// TwinCAT 3 PLC project plc_las_bts_vac
// ProgramVersion: 3.1.4023.0
// libraries:
//   L2SI Vacuum Library, * (SLAC)
//   LCLS General, * (SLAC)
//   PMPS, * (SLAC - LCLS)
//   Tc2_Standard, * (Beckhoff Automation GmbH)
//   Tc2_System, * (Beckhoff Automation GmbH)
//   Tc2_Utilities, * (Beckhoff Automation GmbH)
//   Tc3_Module, * (Beckhoff Automation GmbH)
// project tree:
//   DUTs/ E_TransportTube.TcDUT, ST_TransportTubeConfig.TcDUT, ST_TransportTubeDevices.TcDUT, T_TransportTube.TcDUT
//   DUTs/Operations/ E_Op.TcDUT, E_OpStep.TcDUT
//   DUTs/SystemStatusChecks/ E_GaugeCompOp.TcDUT
//   DUTs/SystemStatusChecks/Switchbox/ ST_SBGaugeReadings.TcDUT, ST_SBGaugeReadingsOp.TcDUT, ST_SBPumpStatuses.TcDUT, ST_SBValveStatuses.TcDUT
//   DUTs/SystemStatusChecks/TransportTubes/ ST_TransportTubeOps.TcDUT, ST_TransportTubeStatuses.TcDUT
//   GVLs/ GVL_BTS_VAC.TcGVL, GVL_Constants.TcGVL, GVL_MaintainLaser.TcGVL, GVL_Operation.TcGVL, GVL_TransportTubes.TcGVL
//   / PlcTask.TcTTO
//   POUs/ FB_TransportTube.TcPOU, F_UpdateIO.TcPOU, MAIN.TcPOU, MaintainLaser.TcPOU, Operate.TcPOU
//   POUs/Helpers/ F_Atm.TcPOU, F_GetTransportTube.TcPOU, F_PumpStationTurboPumpInterlock.TcPOU, F_SBVentInterlock.TcPOU
//   POUs/Operations/Abstracts/ FB_MaintainLaserOperation.TcPOU, FB_Operation.TcPOU, FB_TTOperation.TcPOU
//   POUs/Operations/ FB_LaserOn.TcPOU, FB_OpenTransportTube.TcPOU, FB_SlowPumpSwitchbox.TcPOU, FB_SlowVentSwitchbox.TcPOU, FB_VentTransportTube.TcPOU, FB_VentPumpStation.TcPOU, FB_PumpSwitchbox.TcPOU, FB_VentSwitchbox.TcPOU, FB_PumpTransportTube.TcPOU
//   POUs/Operations/MaintainLaser/ FB_SwitchboxIonPumpFailure.TcPOU, FB_SwitchboxRoughingOrTurboPumpFailure.TcPOU
//   POUs/SystemStatusChecks/ F_CompareGauge.TcPOU
//   POUs/SystemStatusChecks/Switchbox/ F_GetSBGaugeReadings.TcPOU, F_GetSBPumpStatuses.TcPOU, F_GetSBValveStatuses.TcPOU, F_SetSBPumpStatuses.TcPOU, F_SetSBValveStatuses.TcPOU, F_VerifySBGaugeReadings.TcPOU, F_VerifySBPumpStatuses.TcPOU, F_VerifySBValveStatuses.TcPOU
//   POUs/SystemStatusChecks/TransportTubes/ F_GetTransportTubeStatuses.TcPOU, F_SetTransportTubeStatuses.TcPOU, F_VerifyAllTransportTubeStatuses.TcPOU, F_VerifyTransportTubeStatuses.TcPOU (not stored)
// real-time tasks:
//   TASK PlcTask: cycle T#10ms, priority 20, ADS port 350
//   TASK OperateTask: cycle T#10ms, priority 22, ADS port 352
// I/O:
//   DEVICE =+-EK1200_00_00-CPU/EtherCAT1 (disabled), AmsNetId 5.66.246.1.2.1
//     =+-EK1200_00_00 [EK1200-5000 EtherCAT Power supply (2A E-Bus)]
//       =+-EL2794_00_01 [EL2794 4Ch. Dig. Output 24V AC/DC, 2A, short-circuit-proof]
//       =+-ES1004_00_02 [EL1004 4Ch. Dig. Input 24V, 3ms]
//       =+-ES3064_00_03 [EL3064 4Ch. Ana. Input 0-10V]
//       =+-EL1004_00_04 [EL1004 4Ch. Dig. Input 24V, 3ms]
//       =+-EL1004_00_05 [EL1004 4Ch. Dig. Input 24V, 3ms]
//       =+-EL2004_00_06 [EL2004 4Ch. Dig. Output 24V, 0.5A]
//       =+-EL1004_00_07 [EL1004 4Ch. Dig. Input 24V, 3ms]
//       =+-EL2004_00_08 [EL2004 4Ch. Dig. Output 24V, 0.5A]
//       =+-EL2004_00_09 [EL2004 4Ch. Dig. Output 24V, 0.5A]
//       =+-EL1004_00_10 [EL1004 4Ch. Dig. Input 24V, 3ms]
//       =+-EL2794_00_11 [EL2794 4Ch. Dig. Output 24V AC/DC, 2A, short-circuit-proof]
//       =+-EL1004_00_12 [EL1004 4Ch. Dig. Input 24V, 3ms]
//       =+-EL2004_00_13 [EL2004 4Ch. Dig. Output 24V, 0.5A]
//       =+-EL6021_00_14 [EL6021 Interface (RS422/485)]
//       =+-EL2202_00_15 [EL2202 2Ch. Dig. Output 24V, 0.5A]
//       =+-EL1008_00_16 [EL1008 8Ch. Dig. Input 24V, 3ms]
//       =+-EL2008_00_17 [EL2008 8Ch. Dig. Output 24V, 0.5A]
//       =+-EK1110_00_18 [EK1110 EtherCAT extension]
//     =+-EK1100_01_00 [EK1100 EtherCAT Coupler (2A E-Bus)]
//       =+-EL3174_01_18 [EL3174-0002 4Ch. Ana. Input +/-10V, +/-20mA 16 Bit, Isolated Channels]
//       =+-EL3174_01_19 [EL3174-0002 4Ch. Ana. Input +/-10V, +/-20mA 16 Bit, Isolated Channels]
//       =+-EL9184_01_20 [EL9184 Potential Connection, 8 x 24V, 8 x Ground]
//       =+-EL9070_01_21 [EL9070 Shield terminal]
//       =+-EL9070_01_22 [EL9070 Shield terminal]
//       =+-EL3174_01_23 [EL3174-0002 4Ch. Ana. Input +/-10V, +/-20mA 16 Bit, Isolated Channels]
//       =+-EL9184_01_24 [EL9184 Potential Connection, 8 x 24V, 8 x Ground]
//       =+-EL2624_01_25 [EL2624 4Ch. Relay Output, NO (125V AC / 30V DC)]
//       =+-EL2624_01_26 [EL2624 4Ch. Relay Output, NO (125V AC / 30V DC)]
//       =+-EL9505_01_27 [EL9505 Power supply terminal 5V]
//       =+-EL1124_01_28 [EL1124 4Ch. Dig. Input 5V, 10µs, Sensor Power]
//       =+-EL1124_01_29 [EL1124 4Ch. Dig. Input 5V, 10µs, Sensor Power]
//       =+-EL1124_01_30 [EL1124 4Ch. Dig. Input 5V, 10µs, Sensor Power]
//       =+-EL9410_01_31 [EL9410 E-Bus Power Supplier  (Diagnostics)]
//       =+-EL1004_01_32 [EL1004 4Ch. Dig. Input 24V, 3ms]
//       =+-EL1004_01_33 [EL1004 4Ch. Dig. Input 24V, 3ms]
//       =+-EL2794_01_34 [EL2794 4Ch. Dig. Output 24V AC/DC, 2A, short-circuit-proof]
//       =+-EK1122_01_35 [EK1122-0080 2 port EtherCAT junction (Fast Hot Connect)]
//       =+-EK1110_01_36 [EK1110 EtherCAT extension]
// variable links:
//   plc_las_bts_vac/plc_las_bts_vac Instance <-> =+-EK1200_00_00-CPU/EtherCAT1/=+-EK1100_01_00/=+-EL1124_01_28
//     PlcTask Inputs/GVL_BTS_VAC.fb_BI1_GCC.i_xDisc_Active <-> Channel 4/fb_BI1_GCC.i_xDisc_Active
//     PlcTask Inputs/GVL_BTS_VAC.fb_BI1_GCC.i_xHV_ON <-> Channel 3/fb_BI1_GCC.i_xHV_ON
//     PlcTask Inputs/GVL_BTS_VAC.fb_PP_GCC.i_xDisc_Active <-> Channel 2/fb_PP_GCC.i_xDisc_Active
//     PlcTask Inputs/GVL_BTS_VAC.fb_PP_GCC.i_xHV_ON <-> Channel 1/fb_PP_GCC.i_xHV_ON
//   plc_las_bts_vac/plc_las_bts_vac Instance <-> =+-EK1200_00_00-CPU/EtherCAT1/=+-EK1100_01_00/=+-EL1124_01_29
//     PlcTask Inputs/GVL_BTS_VAC.fb_BO4_GCC.i_xDisc_Active <-> Channel 2/fb_BO4_GCC.i_xDisc_Active
//     PlcTask Inputs/GVL_BTS_VAC.fb_BO4_GCC.i_xHV_ON <-> Channel 1/fb_BO4_GCC.i_xHV_ON
//     PlcTask Inputs/GVL_BTS_VAC.fb_DP_GCC.i_xDisc_Active <-> Channel 4/fb_DP_GCC.i_xDisc_Active
//     PlcTask Inputs/GVL_BTS_VAC.fb_DP_GCC.i_xHV_ON <-> Channel 3/fb_DP_GCC.i_xHV_ON
//   plc_las_bts_vac/plc_las_bts_vac Instance <-> =+-EK1200_00_00-CPU/EtherCAT1/=+-EK1100_01_00/=+-EL2624_01_26
//     PlcTask Outputs/GVL_BTS_VAC.fb_BI1_GCC.q_xHV_DIS <-> Channel 3/fb_BI1_GCC.q_xHV_DIS
//     PlcTask Outputs/GVL_BTS_VAC.fb_BO4_GCC.q_xHV_DIS <-> Channel 1/fb_BO4_GCC.q_xHV_DIS
//     PlcTask Outputs/GVL_BTS_VAC.fb_DP_GCC.q_xHV_DIS <-> Channel 4/fb_DP_GCC.q_xHV_DIS
//     PlcTask Outputs/GVL_BTS_VAC.fb_PP_GCC.q_xHV_DIS <-> Channel 2/fb_PP_GCC.q_xHV_DIS
//   plc_las_bts_vac/plc_las_bts_vac Instance <-> =+-EK1200_00_00-CPU/EtherCAT1/=+-EK1100_01_00/=+-EL3174_01_18
//     PlcTask Inputs/GVL_BTS_VAC.fb_BI1_GPI.i_iPRESS_R <-> AI Standard Channel 3/fb_BI1_GPI.i_iPRESS_R
//     PlcTask Inputs/GVL_BTS_VAC.fb_BO4_GPI.i_iPRESS_R <-> AI Standard Channel 1/fb_BO4_GPI.i_iPRESS_R
//     PlcTask Inputs/GVL_BTS_VAC.fb_DP_GPI.i_iPRESS_R <-> AI Standard Channel 4/fb_DP_GPI.i_iPRESS_R
//     PlcTask Inputs/GVL_BTS_VAC.fb_PP_GPI_1.i_iPRESS_R <-> AI Standard Channel 2/fb_PP_GPI_1.i_iPRESS_R
//   plc_las_bts_vac/plc_las_bts_vac Instance <-> =+-EK1200_00_00-CPU/EtherCAT1/=+-EK1100_01_00/=+-EL3174_01_19
//     PlcTask Inputs/GVL_BTS_VAC.fb_PP_GPI_2.i_iPRESS_R <-> AI Standard Channel 1/fb_PP_GPI_2.i_iPRESS_R
//   plc_las_bts_vac/plc_las_bts_vac Instance <-> =+-EK1200_00_00-CPU/EtherCAT1/=+-EK1100_01_00/=+-EL3174_01_23
//     PlcTask Inputs/GVL_BTS_VAC.fb_BI1_GCC.i_iPRESS_R <-> AI Standard Channel 3/fb_BI1_GCC.i_iPRESS_R
//     PlcTask Inputs/GVL_BTS_VAC.fb_BO4_GCC.i_iPRESS_R <-> AI Standard Channel 1/fb_BO4_GCC.i_iPRESS_R
//     PlcTask Inputs/GVL_BTS_VAC.fb_DP_GCC.i_iPRESS_R <-> AI Standard Channel 4/fb_DP_GCC.i_iPRESS_R
//     PlcTask Inputs/GVL_BTS_VAC.fb_PP_GCC.i_iPRESS_R <-> AI Standard Channel 2/fb_PP_GCC.i_iPRESS_R
//   plc_las_bts_vac/plc_las_bts_vac Instance <-> =+-EK1200_00_00-CPU/EtherCAT1/=+-EK1200_00_00/=+-EL1004_00_04
//     PlcTask Inputs/GVL_BTS_VAC.fb_BI1_VGC.i_xClsLS <-> Channel 1/fb_BI1_VGC.i_xClsLS
//     PlcTask Inputs/GVL_BTS_VAC.fb_BI1_VGC.i_xOpnLS <-> Channel 2/fb_BI1_VGC.i_xOpnLS
//     PlcTask Inputs/GVL_BTS_VAC.fb_BO4_VGC.i_xClsLS <-> Channel 3/fb_BO4_VGC.i_xClsLS
//     PlcTask Inputs/GVL_BTS_VAC.fb_BO4_VGC.i_xOpnLS <-> Channel 4/fb_BO4_VGC.i_xOpnLS
//   plc_las_bts_vac/plc_las_bts_vac Instance <-> =+-EK1200_00_00-CPU/EtherCAT1/=+-EK1200_00_00/=+-EL1004_00_05
//     PlcTask Inputs/GVL_BTS_VAC.fb_PP_VGC.i_xClsLS <-> Channel 3/fb_PP_VGC.i_xClsLS
//     PlcTask Inputs/GVL_BTS_VAC.fb_PP_VGC.i_xOpnLS <-> Channel 4/fb_PP_VGC.i_xOpnLS
//     PlcTask Inputs/GVL_BTS_VAC.fb_PP_VRC_1.i_xClsLS <-> Channel 1/fb_PP_VRC_1.i_xClsLS
//     PlcTask Inputs/GVL_BTS_VAC.fb_PP_VRC_1.i_xOpnLS <-> Channel 2/fb_PP_VRC_1.i_xOpnLS
//   plc_las_bts_vac/plc_las_bts_vac Instance <-> =+-EK1200_00_00-CPU/EtherCAT1/=+-EK1200_00_00/=+-EL1004_00_07
//     PlcTask Inputs/GVL_BTS_VAC.fb_PP_VRC_2.i_xClsLS <-> Channel 1/fb_PP_VRC_2.i_xClsLS
//     PlcTask Inputs/GVL_BTS_VAC.fb_PP_VRC_3.i_xClsLS <-> Channel 3/fb_PP_VRC_3.i_xClsLS
//     PlcTask Inputs/GVL_BTS_VAC.fb_PP_VRC_2.i_xOpnLS <-> Channel 2/fb_PP_VRC_2.i_xOpnLS
//     PlcTask Inputs/GVL_BTS_VAC.fb_PP_VRC_3.i_xOpnLS <-> Channel 4/fb_PP_VRC_3.i_xOpnLS
//   plc_las_bts_vac/plc_las_bts_vac Instance <-> =+-EK1200_00_00-CPU/EtherCAT1/=+-EK1200_00_00/=+-EL1004_00_10
//     PlcTask Inputs/GVL_BTS_VAC.fb_PP_PMF.i_xAlarm <-> Channel 3/fb_PP_PMF.i_xAlarm
//     PlcTask Inputs/GVL_BTS_VAC.fb_PP_PMF.i_xIsRun <-> Channel 1/fb_PP_PMF.i_xIsRun
//     PlcTask Inputs/GVL_BTS_VAC.fb_PP_PMF.i_xLocal <-> Channel 2/fb_PP_PMF.i_xLocal
//     PlcTask Inputs/GVL_BTS_VAC.fb_PP_PMF.i_xWarning <-> Channel 4/fb_PP_PMF.i_xWarning
//   plc_las_bts_vac/plc_las_bts_vac Instance <-> =+-EK1200_00_00-CPU/EtherCAT1/=+-EK1200_00_00/=+-EL1004_00_12
//     PlcTask Inputs/GVL_BTS_VAC.fb_PP_PTM.i_xAtSpd <-> Channel 1/fb_PP_PTM.i_xAtSpd
//     PlcTask Inputs/GVL_BTS_VAC.fb_PP_PTM.i_xFaultNC <-> Channel 3/fb_PP_PTM.i_xFaultNC
//     PlcTask Inputs/GVL_BTS_VAC.fb_PP_PTM.i_xRemote <-> Channel 2/fb_PP_PTM.i_xRemote
//   plc_las_bts_vac/plc_las_bts_vac Instance <-> =+-EK1200_00_00-CPU/EtherCAT1/=+-EK1200_00_00/=+-EL2004_00_06
//     PlcTask Outputs/GVL_BTS_VAC.fb_BI1_VGC.q_xOPN_DO <-> Channel 1/fb_BI1_VGC.q_xOPN_DO
//     PlcTask Outputs/GVL_BTS_VAC.fb_BO4_VGC.q_xOPN_DO <-> Channel 3/fb_BO4_VGC.q_xOPN_DO
//   plc_las_bts_vac/plc_las_bts_vac Instance <-> =+-EK1200_00_00-CPU/EtherCAT1/=+-EK1200_00_00/=+-EL2004_00_08
//     PlcTask Outputs/GVL_BTS_VAC.fb_PP_VGC.q_xOPN_DO <-> Channel 2/fb_PP_VGC.q_xOPN_DO
//     PlcTask Outputs/GVL_BTS_VAC.fb_PP_VRC_1.q_xOPN_DO <-> Channel 1/fb_PP_VRC_1.q_xOPN_DO
//     PlcTask Outputs/GVL_BTS_VAC.fb_PP_VRC_2.q_xOPN_DO <-> Channel 3/fb_PP_VRC_2.q_xOPN_DO
//     PlcTask Outputs/GVL_BTS_VAC.fb_PP_VRC_3.q_xOPN_DO <-> Channel 4/fb_PP_VRC_3.q_xOPN_DO
//   plc_las_bts_vac/plc_las_bts_vac Instance <-> =+-EK1200_00_00-CPU/EtherCAT1/=+-EK1200_00_00/=+-EL2004_00_09
//     PlcTask Outputs/GVL_BTS_VAC.fb_PP_VVC.q_xOPN_DO <-> Channel 3/fb_PP_VVC.q_xOPN_DO
//     PlcTask Outputs/GVL_BTS_VAC.fb_VP_VVC_1.xCLS_DO <-> Channel 1/fb_VP_VVC_1.xCLS_DO
//     PlcTask Outputs/GVL_BTS_VAC.fb_VP_VVC_2.xCLS_DO <-> Channel 2/fb_VP_VVC_2.xCLS_DO
//   plc_las_bts_vac/plc_las_bts_vac Instance <-> =+-EK1200_00_00-CPU/EtherCAT1/=+-EK1200_00_00/=+-EL2004_00_13
//     PlcTask Outputs/GVL_BTS_VAC.fb_PP_PTM.q_PumpingStation <-> Channel 3/fb_PP_PTM.q_PumpingStation
//     PlcTask Outputs/GVL_BTS_VAC.fb_PP_PTM.q_RunDO <-> Channel 1/fb_PP_PTM.q_RunDO
//     PlcTask Outputs/GVL_BTS_VAC.fb_PP_PTM.q_xRemote <-> Channel 2/fb_PP_PTM.q_xRemote
//   plc_las_bts_vac/plc_las_bts_vac Instance <-> =+-EK1200_00_00-CPU/EtherCAT1/=+-EK1200_00_00/=+-EL2794_00_01
//     PlcTask Outputs/GVL_BTS_VAC.fb_BI1_PIP.q_xHVEna_DO <-> Channel 2/fb_BI1_PIP.q_xHVEna_DO
//     PlcTask Outputs/GVL_BTS_VAC.fb_BO4_PIP.q_xHVEna_DO <-> Channel 1/fb_BO4_PIP.q_xHVEna_DO
//     PlcTask Outputs/GVL_BTS_VAC.fb_PP_PIP.q_xHVEna_DO <-> Channel 3/fb_PP_PIP.q_xHVEna_DO
//   plc_las_bts_vac/plc_las_bts_vac Instance <-> =+-EK1200_00_00-CPU/EtherCAT1/=+-EK1200_00_00/=+-EL2794_00_11
//     PlcTask Outputs/GVL_BTS_VAC.fb_PP_PMF.q_xLspdDo <-> Channel 2/fb_PP_PMF.q_xLspdDo
//     PlcTask Outputs/GVL_BTS_VAC.fb_PP_PMF.q_xResetDo <-> Channel 3/fb_PP_PMF.q_xResetDo
//     PlcTask Outputs/GVL_BTS_VAC.fb_PP_PMF.q_xRunDO <-> Channel 1/fb_PP_PMF.q_xRunDO
//   plc_las_bts_vac/plc_las_bts_vac Instance <-> =+-EK1200_00_00-CPU/EtherCAT1/=+-EK1200_00_00/=+-ES1004_00_02
//     PlcTask Inputs/GVL_BTS_VAC.fb_BI1_PIP.i_xSP_DI <-> Channel 2/fb_BI1_PIP.i_xSP_DI
//     PlcTask Inputs/GVL_BTS_VAC.fb_BO4_PIP.i_xSP_DI <-> Channel 1/fb_BO4_PIP.i_xSP_DI
//     PlcTask Inputs/GVL_BTS_VAC.fb_PP_PIP.i_xSP_DI <-> Channel 3/fb_PP_PIP.i_xSP_DI
//   plc_las_bts_vac/plc_las_bts_vac Instance <-> =+-EK1200_00_00-CPU/EtherCAT1/=+-EK1200_00_00/=+-ES3064_00_03
//     PlcTask Inputs/GVL_BTS_VAC.fb_BI1_PIP.i_iPRESS <-> AI Standard Channel 2/fb_BI1_PIP.i_iPRESS
//     PlcTask Inputs/GVL_BTS_VAC.fb_BO4_PIP.i_iPRESS <-> AI Standard Channel 1/fb_BO4_PIP.i_iPRESS
//     PlcTask Inputs/GVL_BTS_VAC.fb_PP_PIP.i_iPRESS <-> AI Standard Channel 3/fb_PP_PIP.i_iPRESS

CONFIGURATION plc_las_bts_vac
    RESOURCE PLC ON TwinCAT3
        TASK PlcTask(INTERVAL := T#10ms, PRIORITY := 20);
        PROGRAM MAIN WITH PlcTask : MAIN;
        PROGRAM Operate WITH PlcTask : Operate;
        PROGRAM MaintainLaser WITH PlcTask : MaintainLaser;
    END_RESOURCE
END_CONFIGURATION

// ---- DUTs/E_TransportTube.TcDUT
{attribute 'qualified_only'}
TYPE E_TransportTube :
(
	LS1 := 0,
	LS5 := 1,
	LS8 := 2,
	LD2 := 3,
	LD4 := 4,
	LD6 := 5,
	LD8 := 6,
	LD9 := 7,
	LD10 := 8,
	LD14 := 9
) UINT;
END_TYPE

// ---- DUTs/Operations/E_Op.TcDUT
{attribute 'qualified_only'}
{attribute 'strict'}
TYPE E_Op :
(
	NONE := 0, // No operation
	PSB := 1, // Pump switchbox
	VSB := 2, // Vent switchbox
	VPS := 3, // Vent pumping station
	PTT := 4, // Transport tube pump down
	VTT := 5, // Transport tube vent
	LTT := 6, // Turn on laser for transport tube
	SPSB := 7, // Slow Pump Switchbox
	SVSB := 8 // Slow Vent switchbox
	//OTT, // Open transport tube gate valve
);
END_TYPE

// ---- DUTs/Operations/E_OpStep.TcDUT
{attribute 'qualified_only'}
{attribute 'strict'}
TYPE E_OpStep :
(
	IDLE := 0,
	START := 1,
	
	(* Pump Switchbox steps *)
	PSB_OPEN_GATE_VALVE,
	PSB_OPEN_PUMP_STATION_VALVES,
	PSB_ROUGH_CHAMBER,
	PSB_TURBO_CHAMBER,
	PSB_SWITCH_TO_ION_PUMP,
	PSB_CLOSE_GATE_VALVE,
	PSB_STOP_TURBO_PUMP,
	PSB_FINISH,
	
	(* Slow Pump switchbox steps *)
	SPSB_OPEN_GATE_VALVE,
	SPSB_OPEN_PUMP_STATION_VALVES,
	SPSB_ROUGH_CHAMBER,
	SPSB_OPEN_FORELINE_VALVE,
	SPSB_TURBO_CHAMBER,
	SPSB_SWITCH_TO_ION_PUMP,
	SPSB_CLOSE_VALVES,
	SPSB_STOP_TURBO_PUMP,
	SPSB_FINISH,
	
	(* Vent Switchbox steps *)
	VSB_CLOSE_GATE_VALVE,
	VSB_CLOSE_FORELINE_VALVE,
	VSB_TURN_OFF_PUMPS,
	VSB_CLOSE_ORING_VALVE,
	VSB_VENT,
	VSB_CLOSE_VENT,
	VSB_FINISH,
	
	(* Slow Vent Switchbox steps *)
	SVSB_CLOSE_GATE_VALVE,
	SVSB_CLOSE_FORELINE_VALVE,
	SVSB_TURN_OFF_PUMPS,
	SVSB_CLOSE_ORING_VALVE,
	SVSB_VENT,
	SVSB_SLOW_VENT,
	SVSB_CLOSE_VENT,
	SVSB_FINISH,
	
	(* Vent pump station *)
	VPS_VENT,
	VPS_CLOSE_VENT,
	VPS_FINISH,
	
	(* Pump Down Transport Tube *)
	POT_WAIT_PUMP_CART,
	POT_TURN_ON_PUMP,
	POT_FINISH,
	
	(* Vent Transport Tube *)
	VOT_VENT,
	VOT_WAIT_PC,
	VOT_FINISH,
	
	(* Open Transport Tube Gate Valve *)
	OTT_OPEN_VALVE,
	OTT_RUN_PSB,
	OTT_RUN_PTT,
	
	(* Laser Transport Tube On *)
	LTT_RUN_PSB,
	LTT_RUN_PTT,
	
	(* Beam On - Switchbox Ion Pump Failure *)
	BOIP_TURN_OFF_ION_PUMP,
	BOIP_OPEN_SB_VALVE,
	BOIP_HOLD,
	BOIP_CLOSE_TRANSPORT_TUBE_VALVES,
	BOIP_CLOSE_SB_VALVE,
	BOIP_TURN_OFF_PUMPS,
	BOIP_CLOSE_PP_VALVES,
	BOIP_VENT_SB,
	
	(* Beam On - Switchbox Roughing Pump or Turbo Pump Failure *)
	BOPL_TURN_ON_ION_PUMP,
	BOPL_CLOSE_PP_VALVES,
	BOPL_TURN_OFF_PP_PUMPS,
	BOPL_HOLD,
	BOPL_CLOSE_TRANSPORT_TUBE_VALVES,
	BOPL_VENT_SB
);
END_TYPE

// ---- DUTs/ST_TransportTubeConfig.TcDUT
TYPE ST_TransportTubeConfig :
STRUCT
	{attribute 'pytmc' := '
		pv: NAME
		io: i
	'}
	sName : STRING(EPICS_STRING_SIZE);
	
	bInput : BOOL; // True for input tube, false for output tube
	
	stDevices : ST_TransportTubeDevices;
END_STRUCT
END_TYPE

// ---- DUTs/ST_TransportTubeDevices.TcDUT
(* Devices common to all transport tubes. *)
TYPE ST_TransportTubeDevices :
STRUCT
	// Pumps
	refIonPump : REFERENCE TO FB_PIP_GAMMA;
	
	// Valves
	refGateValve : REFERENCE TO FB_VGC;
	
	// Gauges
	refPiraniGauge : REFERENCE TO FB_MKS275;
	refColdCathode : REFERENCE TO FB_MKS500;
END_STRUCT
END_TYPE

// ---- DUTs/SystemStatusChecks/E_GaugeCompOp.TcDUT
(* Comparison operators that can be used to compare gauge readings *)
{attribute 'qualified_only'}
{attribute 'strict'}
TYPE E_GaugeCompOp :
(
	IGNORE, // Ignore the gauge reading
	ATM, // Check that gauge is at atmospheric pressure
	_LTE, // Check that gauge is less than or equal to value
	_GTE, // Check that gauge is greater than or equal to value
	STATE // Check that gauge has a specific state
):= IGNORE;
END_TYPE

// ---- DUTs/SystemStatusChecks/Switchbox/ST_SBGaugeReadings.TcDUT
(* Statuses of the gauges for the switchbox *)
TYPE ST_SBGaugeReadings :
STRUCT
	(* Gauge readings *)
	
	fDPPiraniVal : REAL; // LXLHN:DP:GPI
	eDPPiraniState : E_PressureState;
	
	fDPColdCathodeVal : REAL; // LXLHN:DP:GCC
	eDPColdCathodeState : E_PressureState;
	
	fPumpStationPirani1Val : REAL; // LXLHN:PP:GPI:1
	ePumpStationPirani1State : E_PressureState;
	
	fPumpStationPirani2Val : REAL; // LXLHN:PP:GPI:2
	ePumpStationPirani2State : E_PressureState;
	
	fPumpStationColdCathodeVal : REAL; // LXLHN:PP:GCC
	ePumpStationColdCathodeState : E_PressureState;
END_STRUCT
END_TYPE

// ---- DUTs/SystemStatusChecks/Switchbox/ST_SBGaugeReadingsOp.TcDUT
(* What operations should be used to compare gauge status *)
TYPE ST_SBGaugeReadingsOp :
STRUCT
	eDPPiraniOp : E_GaugeCompOp; // LXLHN:DP:GPI
	eDPColdCathodeOp : E_GaugeCompOp; // LXLHN:DP:GCC
	ePumpStationPirani1Op : E_GaugeCompOp; // LXLHN:PP:GPI:1
	ePumpStationPirani2Op : E_GaugeCompOp; // LXLHN:PP:GPI:2
	ePumpStationColdCathodeOp : E_GaugeCompOp; // LXLHN:PP:GCC
END_STRUCT
END_TYPE

// ---- DUTs/SystemStatusChecks/Switchbox/ST_SBPumpStatuses.TcDUT
(* Statuses of the pumps for the switchbox *)
TYPE ST_SBPumpStatuses :
STRUCT
	// Pump statuses
	bRoughingPumpOn : BOOL; // LXLHN:PP:PMF
	bTurboPumpOn : BOOL; // LXLHN:PP:PTM
	bIonPumpOn : BOOL; // LXLHN:PP:PIP
END_STRUCT
END_TYPE

// ---- DUTs/SystemStatusChecks/Switchbox/ST_SBValveStatuses.TcDUT
(* Statuses of the valves for the switchbox *)
TYPE ST_SBValveStatuses :
STRUCT
	// Valve statuses
	bGateValveOpen : BOOL; // LXLHN:PP:VGC
	bVentValveOpen : BOOL; // LXLHN:PP:VVC
	bORingPumpValveOpen : BOOL; // LXLHN:PP:VRC:1
	bForelineValveOpen : BOOL; // LXLHN:PP:VRC:2
	bSlowPumpValveOpen : BOOL; // LXLHN:PP:VRC:3
	bSBVentOpen : BOOL; // LXLHN:VP:VVC1
	bSBSlowVentOpen : BOOL; // LXLHN:VP:VVC:2
END_STRUCT
END_TYPE

// ---- DUTs/SystemStatusChecks/TransportTubes/ST_TransportTubeOps.TcDUT
TYPE ST_TransportTubeOps :
STRUCT
	// Pumps
	bIonPumpIgnore : BOOL := FALSE;
	
	// Valves
	bGateValveIgnore : BOOL := FALSE;
	
	// Gauges
	ePiraniOp : E_GaugeCompOp := E_GaugeCompOp.IGNORE;
	eColdCathodeOp : E_GaugeCompOp := E_GaugeCompOp.IGNORE;
END_STRUCT
END_TYPE

// ---- DUTs/SystemStatusChecks/TransportTubes/ST_TransportTubeStatuses.TcDUT
(* Statuses of the pumps, valves, and gauges for the for the BO4 Output tube *)
TYPE ST_TransportTubeStatuses :
STRUCT
	// Pump statuses
	bIonPumpOn : BOOL;
	
	// Valve statuses
	bGateValveOpen : BOOL;
	
	// Gauge statuses
	fPiraniVal : REAL;
	ePiraniState : E_PressureState;
	fColdCathodeVal : REAL;
	eColdCathodeState : E_PressureState;
	
END_STRUCT
END_TYPE

// ---- DUTs/T_TransportTube.TcDUT
// Create a generic transport tube type in case E_TransportTube ever needs to be split up into
// multiple enums (such as input and output tubes). That way all the different Transport tube enums 
// can still have a common type.
TYPE T_TransportTube : UINT; END_TYPE

// ---- GVLs/GVL_BTS_VAC.TcGVL
{attribute 'qualified_only'}
VAR_GLOBAL
	(* Valves *)	
	fb_PP_VGC_FFOut : FB_HardwareFFOutput;
	{attribute 'pytmc' := 'pv: LXLHN:PP:VGC'}
	fb_PP_VGC : FB_VGC; // Gate valve, vacuum switchbox
	
	{attribute 'pytmc' := 'pv: LXLHN:PP:VVC'}
	fb_PP_VVC : FB_VVC; // Turbo N2 purge
	
	{attribute 'pytmc' := 'pv: LXLHN:PP:VRC:1'}
	fb_PP_VRC_1 : FB_VRC; // O-ring diff pump valve
	
	{attribute 'pytmc' := 'pv: LXLHN:PP:VRC:2'}
	fb_PP_VRC_2 : FB_VRC; // Foreline valve
	
	{attribute 'pytmc' := 'pv: LXLHN:PP:VRC:3'}
	fb_PP_VRC_3 : FB_VRC; // Slow pump valve
	
	st_VP_VVC_1 : ST_VCC_NO;
	{attribute 'pytmc' := 'pv: LXLHN:VP:VVC:1'}
	fb_VP_VVC_1 : FB_VCC_NO; // Vent valve, Switchbox
	
	st_VP_VVC_2 : ST_VCC_NO;
	{attribute 'pytmc' := 'pv: LXLHN:VP:VVC:2'}
	fb_VP_VVC_2 : FB_VCC_NO; // Vent valve, Slow, Switchbox

	
	(* Pumps *)
	{attribute 'pytmc' := 'pv: LXLHN:PP:PTM'}
	fb_PP_PTM : FB_PTM_Pfeiffer; // Turbo pump
	
	{attribute 'pytmc' := 'pv: LXLHN:PP:PMF'}
	fb_PP_PMF : FB_KashiyamaPump; // Roughing Pump
	
	{attribute 'pytmc' := 'pv: LXLHN:PP:PIP'}
	fb_PP_PIP : FB_PIP_Gamma; // Ion Pump, SW
	
	(* Gauges *)
	{attribute 'pytmc' := 'pv: LXLHN:PP:GPI:1'}
	fb_PP_GPI_1 : FB_MKS275; // Switchbox pumpline ATM gauge
	
	{attribute 'pytmc' := 'pv: LXLHN:PP:GPI:2'}
	fb_PP_GPI_2 : FB_MKS275; // Foreline gauge
	
	{attribute 'pytmc' := 'pv: LXLHN:DP:GPI'}
	fb_DP_GPI : FB_MKS275; // Switchbox gauge
	
	{attribute 'pytmc' := 'pv: LXLHN:PP:GCC'}
	fb_PP_GCC : FB_MKS500; // Switchbox pumpline Cold Cathode gauge
	
	{attribute 'pytmc' := 'pv: LXLHN:DP:GCC'}
	fb_DP_GCC : FB_MKS500; // Switchbox Cold Cathode gauge
	
	(* Transport Tubes *)
	// LS1
	fb_LS1_VGC_FFOut : FB_HardwareFFOutput;
	{attribute 'pytmc' := 'pv: LTLHN:LS1:VGC:01'}
	fb_LS1_VGC : FB_VGC; // Gate valve, Input LS1 laser Table
	{attribute 'pytmc' := 'pv: LTLHN:LS1:PIP:01'}
	fb_LS1_PIP : FB_PIP_Gamma; // Ion Pump, input tube LS1
	{attribute 'pytmc' := 'pv: LTLHN:LS1:GPI:01'}
	fb_LS1_GPI : FB_MKS275; // Input tube LS1 ATM gauge
	{attribute 'pytmc' := 'pv: LTLHN:LS1:GCC:01'}
	fb_LS1_GCC : FB_MKS500; // Input tube LS1, Cold Cathode gauge
	
	// LS5
	fb_LS5_VGC_FFOut : FB_HardwareFFOutput;
	{attribute 'pytmc' := 'pv: LTLHN:LS5:VGC:01'}
	fb_LS5_VGC : FB_VGC; // Gate valve, Input LS5 laser Table
	{attribute 'pytmc' := 'pv: LTLHN:LS5:PIP:01'}
	fb_LS5_PIP : FB_PIP_Gamma; // Ion Pump, input tube LS5
	{attribute 'pytmc' := 'pv: LTLHN:LS5:GPI:01'}
	fb_LS5_GPI : FB_MKS275; // Input tube LS5 ATM gauge
	{attribute 'pytmc' := 'pv: LTLHN:LS5:GCC:01'}
	fb_LS5_GCC : FB_MKS500; // Input tube LS5, Cold Cathode gauge
	
	// LS8
	fb_LS8_VGC_FFOut : FB_HardwareFFOutput;
	{attribute 'pytmc' := 'pv: LTLHN:LS8:VGC:01'}
	fb_LS8_VGC : FB_VGC; // Gate valve, Input LS8 laser Table
	{attribute 'pytmc' := 'pv: LTLHN:LS8:PIP:01'}
	fb_LS8_PIP : FB_PIP_Gamma; // Ion Pump, input tube LS8
	{attribute 'pytmc' := 'pv: LTLHN:LS8:GPI:01'}
	fb_LS8_GPI : FB_MKS275; // Input tube LS8 ATM gauge
	{attribute 'pytmc' := 'pv: LTLHN:LS8:GCC:01'}
	fb_LS8_GCC : FB_MKS500; // Input tube LS8, Cold Cathode gauge

	// LD2
	fb_LD2_VGC_FFOut : FB_HardwareFFOutput;
	{attribute 'pytmc' := 'pv: LTLHN:LD2:VGC:01'}
	fb_LD2_VGC : FB_VGC; // Gate valve, Output tube LD2 laser Table
	{attribute 'pytmc' := 'pv: LTLHN:LD2:PIP:01'}
	fb_LD2_PIP : FB_PIP_Gamma; // Ion Pump, output tube LD2
	{attribute 'pytmc' := 'pv: LTLHN:LD2:GPI:01 '}
	fb_LD2_GPI : FB_MKS275; // Output tube LD2 ATM gauge
	{attribute 'pytmc' := 'pv: LTLHN:LD2:GCC:01'}
	fb_LD2_GCC : FB_MKS500; // Output tube LD2, Cold Cathode gauge
	
	// LD4
	fb_LD4_VGC_FFOut : FB_HardwareFFOutput;
	{attribute 'pytmc' := 'pv: LTLHN:LD4:VGC:01'}
	fb_LD4_VGC : FB_VGC; // Gate valve, Output tube LD4 laser Table
	{attribute 'pytmc' := 'pv: LTLHN:LD4:PIP:01'}
	fb_LD4_PIP : FB_PIP_Gamma; // Ion Pump, output tube LD4
	{attribute 'pytmc' := 'pv: LTLHN:LD4:GPI:01'}
	fb_LD4_GPI : FB_MKS275; // Output tube LD4 ATM gauge
	{attribute 'pytmc' := 'pv: LTLHN:LD4:GCC:01'}
	fb_LD4_GCC : FB_MKS500; // Output tube LD4, Cold Cathode gauge
	
	// LD6
	fb_LD6_VGC_FFOut : FB_HardwareFFOutput;
	{attribute 'pytmc' := 'pv: LTLHN:LD6:VGC:01'}
	fb_LD6_VGC : FB_VGC; // Gate valve, Output tube LD6 laser Table
	{attribute 'pytmc' := 'pv: LTLHN:LD6:PIP:01'}
	fb_LD6_PIP : FB_PIP_Gamma; // Ion Pump, output tube LD6
	{attribute 'pytmc' := 'pv: LTLHN:LD6:GPI:01'}
	fb_LD6_GPI : FB_MKS275; // Output tube LD6 ATM gauge
	{attribute 'pytmc' := 'pv: LTLHN:LD6:GCC:01'}
	fb_LD6_GCC : FB_MKS500; // Output tube LD6, Cold Cathode gauge
	
	// LD14
	fb_LD14_VGC_FFOut : FB_HardwareFFOutput;
	{attribute 'pytmc' := 'pv: LTLHN:LD14:VGC:01'}
	fb_LD14_VGC : FB_VGC; // Gate valve, Output tube LD14 laser Table
	{attribute 'pytmc' := 'pv: LTLHN:LD14:PIP:01'}
	fb_LD14_PIP : FB_PIP_Gamma; // Ion Pump, output tube LD14
	{attribute 'pytmc' := 'pv: LTLHN:LD14:GPI:01'}
	fb_LD14_GPI : FB_MKS275; // Output tube LD14 ATM gauge
	{attribute 'pytmc' := 'pv: LTLHN:LD14:GCC:01'}
	fb_LD14_GCC : FB_MKS500; // Output tube LD14, Cold Cathode gauge
	
	// LD10
	fb_LD10_VGC_FFOut : FB_HardwareFFOutput;
	{attribute 'pytmc' := 'pv: LTLHN:LD10:VGC:01'}
	fb_LD10_VGC : FB_VGC; // Gate valve, Output tube LD10 laser Table
	{attribute 'pytmc' := 'pv: LTLHN:LD10:PIP:01'}
	fb_LD10_PIP : FB_PIP_Gamma; // Ion Pump, output tube LD10
	{attribute 'pytmc' := 'pv: LTLHN:LD10:GPI:01'}
	fb_LD10_GPI : FB_MKS275; // Output tube LD10 ATM gauge
	{attribute 'pytmc' := 'pv: LTLHN:LD10:GCC:01'}
	fb_LD10_GCC : FB_MKS500; // Output tube LD10, Cold Cathode gauge
	
	// LD9
	fb_LD9_VGC_FFOut : FB_HardwareFFOutput;
	{attribute 'pytmc' := 'pv: LTLHN:LD9:VGC:01'}
	fb_LD9_VGC : FB_VGC; // Gate valve, Output tube LD9 laser Table
	{attribute 'pytmc' := 'pv: LTLHN:LD9:PIP:01'}
	fb_LD9_PIP : FB_PIP_Gamma; // Ion Pump, output tube LD9
	{attribute 'pytmc' := 'pv: LTLHN:LD9:GPI:01'}
	fb_LD9_GPI : FB_MKS275; // Output tube LD9 ATM gauge
	{attribute 'pytmc' := 'pv: LTLHN:LD9:GCC:01'}
	fb_LD9_GCC : FB_MKS500; // Output tube LD9, Cold Cathode gauge
	
	// LD8
	fb_LD8_VGC_FFOut : FB_HardwareFFOutput;
	{attribute 'pytmc' := 'pv: LTLHN:LD8:VGC:01'}
	fb_LD8_VGC : FB_VGC; // Gate valve, Output tube LD8 laser Table
	{attribute 'pytmc' := 'pv: LTLHN:LD8:PIP:01'}
	fb_LD8_PIP : FB_PIP_Gamma; // Ion Pump, output tube LD8
	{attribute 'pytmc' := 'pv: LTLHN:LD8:GPI:01'}
	fb_LD8_GPI : FB_MKS275; // Output tube LD8 ATM gauge
	{attribute 'pytmc' := 'pv: LTLHN:LD8:GCC:01'}
	fb_LD8_GCC : FB_MKS500; // Output tube LD8, Cold Cathode gauge

END_VAR

// ---- GVLs/GVL_Constants.TcGVL
VAR_GLOBAL CONSTANT
	ATM_PRESS : INT := 760; // Atmospheric pressure in Torr
	ATM_PRESS_ERR_RNG : INT := 10; // Error range that is still considered atmospheric pressure
	
	EPICS_STRING_SIZE : INT := 40;
	PTM_INTERLOCK_SP : REAL := 1E-2;
END_VAR

// ---- GVLs/GVL_MaintainLaser.TcGVL
{attribute 'qualified_only'}
VAR_GLOBAL
	{attribute 'pytmc' := '
		pv: PLC_LAS_BTS_VAC:LASER_MAINTAINER:BUSY
		io: i
		field: ZNAM NOT_BUSY
		field: ONAM BUSY
	'}
	q_bOperationInProgress : BOOL;
	
	{attribute 'pytmc' := '
		pv: PLC_LAS_BTS_VAC:LASER_MAINTAINER:RESET
		io: o
	'}
	i_bReset : BOOL; // Reset the laser maintainer to default state
	
	{attribute 'pytmc' := '
		pv: PLC_LAS_BTS_VAC:LASER_MAINTAINER:SHUTOFF
		io: o		
	'}
	i_bShutoff : BOOL; // Signal to shutoff all laser ok signals
	
	{attribute 'pytmc' := '
		pv: PLC_LAS_BTS_VAC:LASER_MAINTAINER:ION_PUMP_FAILURE
		io: i
		field: ZNAM OK
		field: ONAM ERROR
		field: OSV MAJOR
	'}
	q_bIonPumpFailure : BOOL;
	
	{attribute 'pytmc' := '
		pv: PLC_LAS_BTS_VAC:LASER_MAINTAINER:TURBO_PUMP_FAILURE
		io: i
		field: ZNAM OK
		field: ONAM ERROR
		field: OSV MAJOR
	'}
	q_bTurboPumpFailure : BOOL;
	
	{attribute 'pytmc' := '
		pv: PLC_LAS_BTS_VAC:LASER_MAINTAINER:ROUGHING_PUMP_FAILURE
		io: i
		field: ZNAM OK
		field: ONAM ERROR
		field: OSV MAJOR
	'}
	q_bRoughingPumpFailure : BOOL;
	
	{attribute 'pytmc' := '
		pv: PLC_LAS_BTS_VAC:LASER_MAINTAINER:MESSAGE
		io: i
	'}
	q_sMessage : STRING(EPICS_STRING_SIZE) := 'No issues';
	
	{attribute 'pytmc' := '
		pv: PLC_LAS_BTS_VAC:LASER_MAINTAINER:SHUTOFF_LATCH
		io: i
		field: ZNAM OK
		field: ONAM LASERS_SHUTOFF
		field: OSV MAJOR
	'}
	q_bShutoffLatch : BOOL;
END_VAR

// ---- GVLs/GVL_Operation.TcGVL
{attribute 'qualified_only'}
VAR_GLOBAL
	// Execute flags for vacuum system operations
	{attribute 'pytmc' := '
		pv: PLC_LAS_BTS_VAC:OPERATION:CANCEL
		io: o
	'}
	i_bCancel : BOOL;
	
	{attribute 'pytmc' := '
		pv: PLC_LAS_BTS_VAC:OPERATION
		io: io
	'}
	iq_eOperation : E_Op;
	
	{attribute 'pytmc' := '
		pv: PLC_LAS_BTS_VAC:OPERATION:TRANSPORT_TUBE
		io: io
	'}
	iq_eTransportTube : E_TransportTube;
	
	{attribute 'pytmc' := '
		pv: PLC_LAS_BTS_VAC:OPERATION:BUSY
		io: i
		field: ZNAM NOT_BUSY
		field: ONAM BUSY
	'}
	q_bBusy : BOOL;
	
	{attribute 'pytmc' := '
		pv: PLC_LAS_BTS_VAC:OPERATION:ERROR
		io: i
		field: ZNAM OK
		field: ONAM ERROR
		field: ZSV NO_ALARM
		field: OSV MAJOR
	'}
	q_bError : BOOL;
	
	{attribute 'pytmc' := '
		pv: PLC_LAS_BTS_VAC:OPERATION:MESSAGE
		io: i
	'}
	q_sMessage : STRING(EPICS_STRING_SIZE);
END_VAR

// ---- GVLs/GVL_TransportTubes.TcGVL
{attribute 'qualified_only'}
VAR_GLOBAL CONSTANT
	// When adding transport tubes make sure to update F_GetTransportTube!
	
	NUM_TRANSPORT_TUBES : UINT := 10;
	
	aTubes : ARRAY [1..NUM_TRANSPORT_TUBES] OF T_TransportTube := [
		(* Input transport tubes *)
		E_TransportTube.LS1,
		E_TransportTube.LS5,
		E_TransportTube.LS8, 
		
		(* Output transport tubes *)
		E_TransportTube.LD2,
		E_TransportTube.LD4,
		E_TransportTube.LD6,
		E_TransportTube.LD8,
		E_TransportTube.LD9,
		E_TransportTube.LD10,
		E_TransportTube.LD14
	];
	
	(* Transport tube configs *)
	
	stLS1 : ST_TransportTubeConfig := (
		sName:= 'LS1',
		bInput := TRUE,
		stDevices:= (
			refIonPump := GVL_BTS_VAC.fb_LS1_PIP,
			refGateValve := GVL_BTS_VAC.fb_LS1_VGC,
			refPiraniGauge := GVL_BTS_VAC.fb_LS1_GPI,
			refColdCathode := GVL_BTS_VAC.fb_LS1_GCC)
	);
	
	stLS5 : ST_TransportTubeConfig := (
		sName:= 'LS5',
		bInput := TRUE,
		stDevices:= (
			refIonPump := GVL_BTS_VAC.fb_LS5_PIP,
			refGateValve := GVL_BTS_VAC.fb_LS5_VGC,
			refPiraniGauge := GVL_BTS_VAC.fb_LS5_GPI,
			refColdCathode := GVL_BTS_VAC.fb_LS5_GCC)
	);
	
	stLS8 : ST_TransportTubeConfig := (
		sName:= 'LS8',
		bInput := TRUE,
		stDevices:= (
			refIonPump := GVL_BTS_VAC.fb_LS8_PIP,
			refGateValve := GVL_BTS_VAC.fb_LS8_VGC,
			refPiraniGauge := GVL_BTS_VAC.fb_LS8_GPI,
			refColdCathode := GVL_BTS_VAC.fb_LS8_GCC)
	);	
	
	stLD2 : ST_TransportTubeConfig := (
		sName:= 'LD2',
		bInput := FALSE,
		stDevices:= (
			refIonPump := GVL_BTS_VAC.fb_LD2_PIP,
			refGateValve := GVL_BTS_VAC.fb_LD2_VGC,
			refPiraniGauge := GVL_BTS_VAC.fb_LD2_GPI,
			refColdCathode := GVL_BTS_VAC.fb_LD2_GCC)
	);
	
	stLD4 : ST_TransportTubeConfig := (
		sName:= 'LD4',
		bInput := FALSE,
		stDevices:= (
			refIonPump := GVL_BTS_VAC.fb_LD4_PIP,
			refGateValve := GVL_BTS_VAC.fb_LD4_VGC,
			refPiraniGauge := GVL_BTS_VAC.fb_LD4_GPI,
			refColdCathode := GVL_BTS_VAC.fb_LD4_GCC)
	);
	
	stLD6 : ST_TransportTubeConfig := (
		sName:= 'LD6',
		bInput := FALSE,
		stDevices:= (
			refIonPump := GVL_BTS_VAC.fb_LD6_PIP,
			refGateValve := GVL_BTS_VAC.fb_LD6_VGC,
			refPiraniGauge := GVL_BTS_VAC.fb_LD6_GPI,
			refColdCathode := GVL_BTS_VAC.fb_LD6_GCC)
	);
	
	stLD14 : ST_TransportTubeConfig := (
		sName:= 'LD14',
		bInput := FALSE,
		stDevices:= (
			refIonPump := GVL_BTS_VAC.fb_LD14_PIP,
			refGateValve := GVL_BTS_VAC.fb_LD14_VGC,
			refPiraniGauge := GVL_BTS_VAC.fb_LD14_GPI,
			refColdCathode := GVL_BTS_VAC.fb_LD14_GCC)
	);
	
	stLD10 : ST_TransportTubeConfig := (
		sName:= 'LD10',
		bInput := FALSE,
		stDevices:= (
			refIonPump := GVL_BTS_VAC.fb_LD10_PIP,
			refGateValve := GVL_BTS_VAC.fb_LD10_VGC,
			refPiraniGauge := GVL_BTS_VAC.fb_LD10_GPI,
			refColdCathode := GVL_BTS_VAC.fb_LD10_GCC)
	);
	
	stLD9 : ST_TransportTubeConfig := (
		sName:= 'LD9',
		bInput := FALSE,
		stDevices:= (
			refIonPump := GVL_BTS_VAC.fb_LD9_PIP,
			refGateValve := GVL_BTS_VAC.fb_LD9_VGC,
			refPiraniGauge := GVL_BTS_VAC.fb_LD9_GPI,
			refColdCathode := GVL_BTS_VAC.fb_LD9_GCC)
	);
	
	stLD8 : ST_TransportTubeConfig := (
		sName:= 'LD8',
		bInput := FALSE,
		stDevices:= (
			refIonPump := GVL_BTS_VAC.fb_LD8_PIP,
			refGateValve := GVL_BTS_VAC.fb_LD8_VGC,
			refPiraniGauge := GVL_BTS_VAC.fb_LD8_GPI,
			refColdCathode := GVL_BTS_VAC.fb_LD8_GCC)
	);

END_VAR
VAR_GLOBAL
	{attribute 'pytmc' := '
		pv: LTLHN:LS1
	'}
	fbLS1 : FB_TransportTube;
	{attribute 'pytmc' := '
		pv: LTLHN:LS5
	'}
	fbLS5 : FB_TransportTube;
	{attribute 'pytmc' := '
		pv: LTLHN:LS8
	'}
	fbLS8 : FB_TransportTube;

	{attribute 'pytmc' := '
		pv: LTLHN:LD2
	'}
	fbLD2 : FB_TransportTube;
	{attribute 'pytmc' := '
		pv: LTLHN:LD4
	'}
	fbLD4 : FB_TransportTube;
	{attribute 'pytmc' := '
		pv: LTLHN:LD6
	'}
	fbLD6 : FB_TransportTube;
	{attribute 'pytmc' := '
		pv: LTLHN:LD14
	'}
	fbLD14 : FB_TransportTube;
	{attribute 'pytmc' := '
		pv: LTLHN:LD10
	'}
	fbLD10 : FB_TransportTube;
	{attribute 'pytmc' := '
		pv: LTLHN:LD9
	'}
	fbLD9 : FB_TransportTube;
	{attribute 'pytmc' := '
		pv: LTLHN:LD8
	'}
	fbLD8 : FB_TransportTube;

END_VAR

// ---- POUs/MAIN.TcPOU
PROGRAM MAIN
VAR
END_VAR

(* Update physical IO signals *)
F_UpdateIO();

(* Update transport tubes *)
GVL_TransportTubes.fbLS1(
	i_stConfig := GVL_TransportTubes.stLS1, 
	i_bLaserExtIntl := TRUE
);

GVL_TransportTubes.fbLS5(
	i_stConfig := GVL_TransportTubes.stLS5, 
	i_bLaserExtIntl := TRUE
);

GVL_TransportTubes.fbLS8(
	i_stConfig := GVL_TransportTubes.stLS8, 
	i_bLaserExtIntl := TRUE
);

GVL_TransportTubes.fbLD2(
	i_stConfig := GVL_TransportTubes.stLD2,
	i_bLaserExtIntl := TRUE
);

GVL_TransportTubes.fbLD4(
	i_stConfig := GVL_TransportTubes.stLD4,
	i_bLaserExtIntl := TRUE
);

GVL_TransportTubes.fbLD6(
	i_stConfig := GVL_TransportTubes.stLD6,
	i_bLaserExtIntl := TRUE
);

GVL_TransportTubes.fbLD14(
	i_stConfig := GVL_TransportTubes.stLD14,
	i_bLaserExtIntl := TRUE
);

GVL_TransportTubes.fbLD10(
	i_stConfig := GVL_TransportTubes.stLD10,
	i_bLaserExtIntl := TRUE
);

GVL_TransportTubes.fbLD9(
	i_stConfig := GVL_TransportTubes.stLD9,
	i_bLaserExtIntl := TRUE
);

GVL_TransportTubes.fbLD8(
	i_stConfig := GVL_TransportTubes.stLD8,
	i_bLaserExtIntl := TRUE
);

END_PROGRAM

// ---- POUs/F_UpdateIO.TcPOU
FUNCTION F_UpdateIO : BOOL
VAR_INPUT
END_VAR
VAR
END_VAR

(* Update Gauges *)
GVL_BTS_VAC.fb_PP_GPI_1();

GVL_BTS_VAC.fb_PP_GPI_2();

GVL_BTS_VAC.fb_DP_GPI();

GVL_BTS_VAC.fb_BO4_GPI();

GVL_BTS_VAC.fb_BI1_GPI();

GVL_BTS_VAC.fb_PP_GCC(PG := GVL_BTS_VAC.fb_PP_GPI_1.PG);

GVL_BTS_VAC.fb_BO4_GCC(PG := GVL_BTS_VAC.fb_BO4_GPI.PG);

GVL_BTS_VAC.fb_BI1_GCC(PG := GVL_BTS_VAC.fb_BI1_GPI.PG);

GVL_BTS_VAC.fb_DP_GCC(PG := GVL_BTS_VAC.fb_DP_GPI.PG);

(* Update vacuum gauge controllers *)
GVL_BTS_VAC.fb_BO4_VGC(
	i_stUSG := GVL_BTS_VAC.fb_BO4_GCC.IG,
	i_stDSG := GVL_BTS_VAC.fb_DP_GCC.IG,
	i_xEPS_OK := TRUE,
	i_xPMPS_OK := TRUE,
	i_xExt_OK := TRUE,
	io_fbFFHWO := GVL_BTS_VAC.fb_BO4_VGC_FFOut
);

GVL_BTS_VAC.fb_PP_VGC(
	i_stUSG := GVL_BTS_VAC.fb_PP_GCC.IG,
	i_stDSG := GVL_BTS_VAC.fb_DP_GCC.IG,
	i_xDis_DPIlk := FALSE,
	i_xEPS_OK := TRUE,
	i_xPMPS_OK := TRUE,
	i_xExt_OK := GVL_BTS_VAC.fb_PP_PTM.iq_stPTM.eState = E_PumpState.pumpRUNNING,
	io_fbFFHWO := GVL_BTS_VAC.fb_PP_VGC_FFOut
);

GVL_BTS_VAC.fb_PP_VVC(
	i_xExtILK_OK := 
		GVL_BTS_VAC.fb_PP_PTM.iq_stPTM.eState = E_PumpState.pumpSTOPPED
		AND GVL_BTS_VAC.fb_PP_VGC.M_IsClosed()
);

GVL_BTS_VAC.fb_PP_VRC_1(
	i_xExtILK_OK := GVL_BTS_VAC.fb_PP_PMF.q_stPump.eState = E_PumpState.pumpRUNNING
);

GVL_BTS_VAC.fb_PP_VRC_2(
	i_xExtILK_OK := GVL_BTS_VAC.fb_PP_PMF.q_stPump.eState = E_PumpState.pumpRUNNING
);

GVL_BTS_VAC.fb_PP_VRC_3(
	i_xExtILK_OK := GVL_BTS_VAC.fb_PP_PMF.q_stPump.eState = E_PumpState.pumpRUNNING
);

GVL_BTS_VAC.fb_BI1_VGC(
	i_stUSG := GVL_BTS_VAC.fb_BI1_GCC.IG, 
	i_stDSG := GVL_BTS_VAC.fb_DP_GCC.IG,
	i_xDis_DPIlk := FALSE,
	i_xEPS_OK := TRUE,
	i_xPMPS_OK := TRUE,
	i_xExt_OK := TRUE,
	io_fbFFHWO := GVL_BTS_VAC.fb_BI1_VGC_FFOut
);

GVL_BTS_VAC.fb_VP_VVC_1(
	iq_stValve := GVL_BTS_VAC.st_VP_VVC_1,
	i_xExtILK_OK := F_SBVentInterlock()
);

GVL_BTS_VAC.fb_VP_VVC_2(
	iq_stValve := GVL_BTS_VAC.st_VP_VVC_2,
	i_xExtILK_OK := F_SBVentInterlock()
);

(* Update pumps *)
GVL_BTS_VAC.fb_PP_PMF();

GVL_BTS_VAC.fb_PP_PTM(i_xExtRunOk := F_PumpStationTurboPumpInterlock());

GVL_BTS_VAC.fb_BO4_PIP(i_stGauge := GVL_BTS_VAC.fb_BO4_GCC.IG);

GVL_BTS_VAC.fb_PP_PIP(i_stGauge := GVL_BTS_VAC.fb_DP_GCC.IG);

GVL_BTS_VAC.fb_BI1_PIP(i_stGauge := GVL_BTS_VAC.fb_BI1_GCC.IG);

END_FUNCTION

// ---- POUs/Helpers/F_SBVentInterlock.TcPOU
// Verify that all Switchbox valves are closed
FUNCTION F_SBVentInterlock : BOOL
VAR_INPUT
END_VAR
VAR
	stExpValveStatus : ST_SBValveStatuses := (
		bGateValveOpen:= FALSE, 
		bVentValveOpen:= FALSE, 
		bORingPumpValveOpen:= FALSE, 
		bForelineValveOpen:= FALSE, 
		bSlowPumpValveOpen:= FALSE,
		bSBVentOpen:= NOT GVL_BTS_VAC.st_VP_VVC_1.xCLS_DO,
		bSBSlowVentOpen:= NOT GVL_BTS_VAC.st_VP_VVC_2.xCLS_DO);
END_VAR

F_SBVentInterlock := F_VerifySBValveStatuses(stExpStatus := stExpValveStatus, bEnforce := FALSE);

END_FUNCTION

// ---- POUs/SystemStatusChecks/Switchbox/F_VerifySBValveStatuses.TcPOU
(* Verify that the statuses of the switchbox valves match the expected statuses *)
FUNCTION F_VerifySBValveStatuses : BOOL
VAR_INPUT
	stExpStatus : ST_SBValveStatuses; // The expected state of the system
	bEnforce : BOOL; // Whether to try forcing the states
END_VAR
VAR
	stStatus : ST_SBValveStatuses;
END_VAR

stStatus := F_GetSBValveStatuses();

IF bEnforce THEN
	// Try setting system states to the expected states
	F_SetSBValveStatuses(stExpStatus);
END_IF

// Return true if the expected status matches the actual status
F_VerifySBValveStatuses := stExpStatus.bGateValveOpen = stStatus.bGateValveOpen
	AND stExpStatus.bVentValveOpen = stStatus.bVentValveOpen
	AND stExpStatus.bORingPumpValveOpen = stStatus.bORingPumpValveOpen
	AND stExpStatus.bForelineValveOpen = stStatus.bForelineValveOpen
	AND stExpStatus.bSBVentOpen = stStatus.bSBVentOpen
	AND stExpStatus.bSlowPumpValveOpen = stStatus.bSlowPumpValveOpen
	AND stExpStatus.bSBSlowVentOpen = stStatus.bSBSlowVentOpen;

END_FUNCTION

// ---- POUs/SystemStatusChecks/Switchbox/F_GetSBValveStatuses.TcPOU
FUNCTION F_GetSBValveStatuses : ST_SBValveStatuses
VAR_INPUT
END_VAR
VAR
	stStatus : ST_SBValveStatuses := (
		bGateValveOpen:= GVL_BTS_VAC.fb_PP_VGC.M_IsOpen(), 
		bVentValveOpen:= GVL_BTS_VAC.fb_PP_VVC.M_IsOpen(), 
		bORingPumpValveOpen:= GVL_BTS_VAC.fb_PP_VRC_1.iq_stValve.eState = E_ValvePositionState.OPEN, 
		bForelineValveOpen:= GVL_BTS_VAC.fb_PP_VRC_2.iq_stValve.eState = E_ValvePositionState.OPEN, 
		bSBVentOpen:= NOT GVL_BTS_VAC.st_VP_VVC_1.xCLS_DO, 
		bSlowPumpValveOpen:= GVL_BTS_VAC.fb_PP_VRC_3.iq_stValve.eState = E_ValvePositionState.OPEN, 
		bSBSlowVentOpen:= NOT GVL_BTS_VAC.st_VP_VVC_2.xCLS_DO);
END_VAR

F_GetSBValveStatuses := stStatus;

END_FUNCTION

// ---- POUs/SystemStatusChecks/Switchbox/F_SetSBValveStatuses.TcPOU
FUNCTION F_SetSBValveStatuses : BOOL
VAR_INPUT
	stExpStatuses : ST_SBValveStatuses;
END_VAR
VAR
END_VAR

GVL_BTS_VAC.fb_PP_VGC.M_Set_OPN_SW(stExpStatuses.bGateValveOpen);
GVL_BTS_VAC.fb_PP_VVC.M_Open(stExpStatuses.bVentValveOpen);
GVL_BTS_VAC.fb_PP_VRC_1.M_Set_OPN_SW(stExpStatuses.bORingPumpValveOpen); 
GVL_BTS_VAC.fb_PP_VRC_2.M_Set_OPN_SW(stExpStatuses.bForelineValveOpen);
GVL_BTS_VAC.fb_PP_VRC_3.M_Set_OPN_SW(stExpStatuses.bSBSlowVentOpen);
GVL_BTS_VAC.fb_VP_VVC_1.M_Close(NOT stExpStatuses.bSBVentOpen);
GVL_BTS_VAC.fb_VP_VVC_2.M_Close(NOT stExpStatuses.bSBSlowVentOpen);

END_FUNCTION

// ---- POUs/Helpers/F_PumpStationTurboPumpInterlock.TcPOU
FUNCTION F_PumpStationTurboPumpInterlock : BOOL
VAR_INPUT
END_VAR
VAR
END_VAR

F_PumpStationTurboPumpInterlock := F_CompareGauge(eCompOp:= E_GaugeCompOp._LTE, fReading:=
										GVL_BTS_VAC.fb_PP_GPI_1.PG.rPRESS, 
										eState:= 0, 
										fExpReading:= PTM_INTERLOCK_SP, 
										eExpState:= 0)
									AND F_CompareGauge(eCompOp:= E_GaugeCompOp._LTE, fReading:=
										GVL_BTS_VAC.fb_PP_GPI_2.PG.rPRESS, 
										eState:= 0, 
										fExpReading:= PTM_INTERLOCK_SP, 
										eExpState:= 0)
									AND GVL_BTS_VAC.fb_PP_VVC.M_IsClosed()
									AND GVL_BTS_VAC.fb_PP_PMF.q_stPump.eState = E_PumpState.pumpRUNNING;

END_FUNCTION

// ---- POUs/SystemStatusChecks/F_CompareGauge.TcPOU
FUNCTION F_CompareGauge : BOOL
VAR_INPUT
	eCompOp : E_GaugeCompOp; // Which compare operation to use
	fReading : REAL; // The actual reading
	eState : E_PressureState; // The actual state the gauge is in
	fExpReading : REAL; // Used to find expected reading
	eExpState : E_PressureState; // The expected state the gauge should be in
END_VAR
VAR
END_VAR

CASE eCompOp OF
E_GaugeCompOp.ATM: // Check the gauge is within atmoshperic pressure range
	F_CompareGauge := F_Atm(fReading);
E_GaugeCompOp._GTE: // Check the gauge is greater than or equal to the expected value
	F_CompareGauge := fReading >= fExpReading;
E_GaugeCompOp._LTE: // Check the gauge is less than or equal to the expected value
	F_CompareGauge := fReading <= fExpReading;
E_GaugeCompOp.STATE: // Check the gauge has the expected state
	F_CompareGauge := eState = eExpState;
E_GaugeCompOp.IGNORE: // Ignore gauge reading
	F_CompareGauge := TRUE;
ELSE // Unimplimented operation
	F_CompareGauge := FALSE;
END_CASE

END_FUNCTION

// ---- POUs/Helpers/F_Atm.TcPOU
// Verifies if a pressure (TORR) is near atmospheric pressure
FUNCTION F_Atm : BOOL
VAR_INPUT
	fPressure : REAL;
END_VAR
VAR
END_VAR

// Check that fPressure is within our error range for atmospheric pressure
F_Atm := ABS(ATM_PRESS - fPressure) <= ATM_PRESS_ERR_RNG;

END_FUNCTION

// ---- POUs/Operate.TcPOU
PROGRAM Operate
VAR
	eCurrOp : E_Op; // The currently running operation
	eCurrTransportTube : T_TransportTube; // The current transport tube being operated on (if operation involves transport tube)
	
	(* Operations *)
	fbPumpTransportTube : FB_PumpTransportTube;
	fbVentTransportTube : FB_VentTransportTube;
	//fbOpenTransportTube : FB_OpenTransportTube;
	fbLaseron : FB_LaserOn;
	fbPumpSwitchbox : FB_PumpSwitchbox;
	fbSlowPumpSwitchbox : FB_SlowPumpSwitchbox;
	fbVentPumpStation : FB_VentPumpStation;
	fbVentSwitchbox : FB_VentSwitchbox;
	fbSlowVentSwitchbox : FB_SlowVentSwitchbox;
END_VAR

(* Run operations, but don't start any new operations if another operation is still running *)

// If the maintain laser program is running an operation, prevent this program from running operations.
IF GVL_MaintainLaser.q_bOperationInProgress THEN
	GVL_Operation.i_bCancel := TRUE;
END_IF

// Only start new operations if the system is NOT busy with another operation!
IF NOT GVL_Operation.q_bBusy THEN
	eCurrOp := GVL_Operation.iq_eOperation;
	eCurrTransportTube := GVL_Operation.iq_eTransportTube;
END_IF

// Execute selected operation
CASE eCurrOp OF
E_Op.NONE: // No operation selected
	GVL_Operation.q_bBusy := FALSE;

E_Op.PTT: // Pump transport tube
	fbPumpTransportTube(
		i_bExecute := TRUE, 
		i_bCancel := GVL_Operation.i_bCancel,
		iq_sMessageBuffer := GVL_Operation.q_sMessage,
		i_eTransportTube := eCurrTransportTube,
		q_bBusy => GVL_Operation.q_bBusy,
		q_bError => GVL_Operation.q_bError
	);

E_Op.VTT: // Vent transport tube
	fbVentTransportTube(
		i_bExecute := TRUE,
		i_bCancel := GVL_Operation.i_bCancel,
		iq_sMessageBuffer := GVL_Operation.q_sMessage,
		i_eTransportTube := eCurrTransportTube,
		q_bBusy => GVL_Operation.q_bBusy,
		q_bError => GVL_Operation.q_bError
	);
	
(*
E_Op.OTT: // Open transport tube gate valve
	fbOpenTransportTube(
		i_bExecute := TRUE,
		i_bCancel := i_bCancel,
		iq_sMessageBuffer := GVL_Operation.q_sMessage,
		i_eTransportTube := eCurrTransportTube,
		q_bBusy => GVL_Operation.q_bBusy,
		q_bError => GVL_Operation.q_bError
	);
*)
	
E_Op.LTT: // Turn laser on for transport tube
	fbLaserOn(
		i_bExecute := TRUE,
		i_bCancel := GVL_Operation.i_bCancel,
		iq_sMessageBuffer := GVL_Operation.q_sMessage,
		i_eTransporttube := eCurrTransportTube,
		q_bBusy => GVL_Operation.q_bBusy,
		q_bError => GVL_Operation.q_bError
	);
	
E_Op.PSB: // Pump switchbox
	fbPumpSwitchbox(
		i_bExecute := TRUE,
		i_bCancel := GVL_Operation.i_bCancel,
		iq_sMessageBuffer := GVL_Operation.q_sMessage,
		q_bBusy => GVL_Operation.q_bBusy,
		q_bError => GVL_Operation.q_bError
	);
	
E_Op.SPSB: // Slow pump switchbox
	fbSlowPumpSwitchbox(
		i_bExecute := TRUE,
		i_bCancel := GVL_Operation.i_bCancel,
		iq_sMessageBuffer := GVL_Operation.q_sMessage,
		q_bBusy => GVL_Operation.q_bBusy,
		q_bError => GVL_Operation.q_bError
	);
	
E_Op.VPS: // Vent pump station
	fbVentPumpStation(
		i_bExecute := TRUE,
		i_bCancel := GVL_Operation.i_bCancel,
		iq_sMessageBuffer := GVL_Operation.q_sMessage,
		q_bBusy => GVL_Operation.q_bBusy,
		q_bError => GVL_Operation.q_bError
	);

E_Op.VSB: // Vent switchbox
	fbVentSwitchbox(
		i_bExecute := TRUE,
		i_bCancel := GVL_Operation.i_bCancel,
		iq_sMessageBuffer := GVL_Operation.q_sMessage,
		q_bBusy => GVL_Operation.q_bBusy,
		q_bError => GVL_Operation.q_bError
	);
	
E_Op.SVSB: // Slow vent switchbox
	fbSlowVentSwitchbox(
		i_bExecute := TRUE,
		i_bCancel := GVL_Operation.i_bCancel,
		iq_sMessageBuffer := GVL_Operation.q_sMessage,
		q_bBusy => GVL_Operation.q_bBusy,
		q_bError => GVL_Operation.q_bError
	);
	
ELSE // Operator selected unimplemented operation
	GVL_Operation.q_sMessage := 'Unimplemented operation';
	GVL_Operation.q_bBusy := FALSE;
	GVL_Operation.q_bError := TRUE;
END_CASE

// If all operation have finished then set operation back to none
IF NOT GVL_Operation.q_bBusy THEN
	eCurrOp := E_Op.NONE;
END_IF

// Set output operation to whatever is ACTAULLY currently running
GVL_Operation.iq_eOperation := eCurrOp;
GVL_Operation.iq_eTransportTube := eCurrTransportTube;
GVL_Operation.i_bCancel := FALSE; // Reset cancel flag

END_PROGRAM

// ---- POUs/Operations/FB_PumpTransportTube.TcPOU
FUNCTION_BLOCK FB_PumpTransportTube EXTENDS FB_TTOperation
VAR_STAT CONSTANT
	(* Expected system states before operation starts*)		
	stExpTTStatus : ST_TransportTubeStatuses := (
		bIonPumpOn:= FALSE,
		bGateValveOpen:= FALSE,
		eColdCathodeState:= E_PressureState.Off);
	stTTOp : ST_TransportTubeOps := (
		ePiraniOp := E_GaugeCompOp.ATM,
		eColdCathodeOp := E_GaugeCompOp.STATE
	);
		
	(* Expected system states after operation finishes *)		
	stFinExpTTStatus : ST_TransportTubeStatuses := (
		bIonPumpOn:= TRUE,
		bGateValveOpen:= FALSE,
		ePiraniState:= E_PressureState.ValidLo,
		fColdCathodeVal:= 1E-5);
	stFinTTOp : ST_TransportTubeOps := (
		ePiraniOp := E_GaugeCompOp.STATE,
		eColdCathodeOp := E_GaugeCompOp._LTE
	);
		
	(* Timeout constants *);
	PUMP_CART_TIMEOUT : TIME := T#20M;
	ION_PUMP_TIMEOUT : TIME := T#15M;
	
	(* Pressure constants *)
	ION_READY_PRESS : REAL := 1E-4; // Pressure at which to initiate ion pump
	ION_FINISHED_PRESS : REAL := 1E-5; // Pressure at which pressure has reached desired state
END_VAR

SUPER^(iq_sMessageBuffer := iq_sMessageBuffer);

CASE eStep OF
E_OpStep.IDLE: // Do nothing

E_OpStep.START: // Verify system status
	M_RunTimeoutTimer(STATUS_CHECK_TIMEOUT);
	
	M_SetMessage('Verifying system status');
	
	IF F_VerifyTransportTubeStatuses(stExpStatus := stExpTTStatus,
		eTransportTube := eTT,
		stStatusOp := stTTOp, 
		bEnforce := TRUE)
	THEN // System status check 
		M_ResetTimeoutTimer();
		M_SetMessage('OPERATOR: Rough chamber w/ pump cart'); 
		eStep := E_OpStep.POT_WAIT_PUMP_CART;
	END_IF
	
E_OpStep.POT_WAIT_PUMP_CART:
	M_RunTimeoutTimer(PUMP_CART_TIMEOUT);
	(* At this point the system must wait for the transport tube to be roughed by the pump cart.
	   The pump cart is manually operated, so we will wait until the desired pressure is reached.
	*)
	
	// Check that pressure is low enough to turn on ion pump
	IF fbTT.q_stConfig.stDevices.refPiraniGauge.PG.rPRESS <= ION_READY_PRESS THEN
		M_ResetTimeoutTimer();
		M_SetMessage('Turning on ion pump');
		eStep := E_OpStep.POT_TURN_ON_PUMP;
	END_IF
	
E_OpStep.POT_TURN_ON_PUMP:
	M_RunTimeoutTimer(ION_PUMP_TIMEOUT);
	
	fbTT.q_stConfig.stDevices.refIonPump.M_Run(TRUE);
	// Check that desired pressure has been reached
	IF fbTT.q_stConfig.stDevices.refColdCathode.IG.eState <> E_PressureState.Off
	AND fbTT.q_stConfig.stDevices.refColdCathode.IG.rPRESS <= ION_FINISHED_PRESS
	THEN
		M_ResetTimeoutTimer();
		eStep := E_OpStep.POT_FINISH;
	END_IF
	
E_OpStep.POT_FINISH:
	IF F_VerifyTransportTubeStatuses(stExpStatus := stFinExpTTStatus,
		eTransportTube := eTT,
		stStatusOp := stFinTTOp, 
		bEnforce := FALSE)
	THEN
		M_Finish();
	ELSE
		M_FatalError('End system status check failed');
	END_IF
	
ELSE
	M_FatalError('Operation is in invalid state');
END_CASE

END_FUNCTION_BLOCK

// ---- POUs/Operations/Abstracts/FB_TTOperation.TcPOU
// Operate on a transport tube
FUNCTION_BLOCK FB_TTOperation EXTENDS FB_Operation
VAR_INPUT
	i_eTransportTube : T_TransportTube;
END_VAR
VAR
	fbTT : REFERENCE TO FB_TransportTube;
	eTT : T_TransportTube; 
END_VAR

// If going from idle to starting a new operation then update the transport tube reference
// We do this before running the parent class because the eStep has not changed yet.
IF eStep = E_OpStep.IDLE AND i_bExecute = TRUE THEN
	eTT := i_eTransportTube; // Copy the input to ensure transport tube doesn't get changed from the outside
	fbTT REF= F_GetTransportTube(eTT);
END_IF;

// Let FB_Operation do its thing 
SUPER^(iq_sMessageBuffer := iq_sMessageBuffer);

// Check that reference to transport tube is valid
// We do this after the parent class has run so that the fatal error does not get overriden
IF eStep <> E_OpStep.IDLE AND NOT __ISVALIDREF(fbTT) THEN
	M_FatalError('Invalid transport tube');
END_IF

END_FUNCTION_BLOCK

// ---- POUs/Operations/Abstracts/FB_Operation.TcPOU
FUNCTION_BLOCK FB_Operation
VAR_INPUT
	i_bExecute : BOOL; // Flag that indicates the operation should be ran
	i_bCancel : BOOL; // Cancel operation input signal
END_VAR
VAR_IN_OUT
	iq_sMessageBuffer : STRING(EPICS_STRING_SIZE); // Human readable description of the current step
END_VAR
VAR_OUTPUT
	q_bError : BOOL; // Whether a fatal error was encountered
	q_bBusy : BOOL; // Whether the current operation is executing
END_VAR
VAR
	bCancel : BOOL; // Saved cancel operation signal
	bDeferCancel : BOOL; // Setting to True prevents operation from being immediatly cancelled with i_bCancel. Resets to FALSE after operation finishes
	eStep : E_OpStep := E_OpStep.IDLE; // The current operation step
	fbTimeoutTimer : TON; // TImer used for tracking operation timeouts
END_VAR
VAR_STAT CONSTANT
	STATUS_CHECK_TIMEOUT : TIME := T#30S; // How long the system tries setting the desired state before failing
	VALVE_TIMEOUT : TIME := T#10S; // How long system tries to open or close valve before failing
	ROUGH_CHAMBER_TIMEOUT : TIME := T#5M; // How long to try rough pumping before failing
	TURBO_CHAMBER_TIMEOUT : TIME := T#10M; // How long to try turbo pumping before failing
	PUMP_TIMEOUT : TIME := T#20S; // How long to try to turn on or off pump before failing
END_VAR

IF eStep = E_OpStep.IDLE AND i_bExecute = TRUE THEN
	// Start operation
	eStep := E_OpStep.START;
	q_bBusy := TRUE;
	M_ResetError();
END_IF

(* Save the input i_bCancel signal since cancelling can take multiple cycles *)
IF i_bCancel THEN
	bCancel := TRUE;
END_IF

(* Allow operation to be cancelled from an input signal.
 The cancel input signal can be deferred by the operation if the 
 operation is not at a good point to finish cancelling. *)
IF eStep <> E_OpStep.IDLE AND NOT bDeferCancel AND bCancel THEN
	M_FatalError('Operation canceled');
END_IF

IF M_TimeoutExpired() THEN // If a timeout has expired, trigger a fatal error
	M_FatalError('Timeout expired');
END_IF

// Defer cancel signals until a later time
METHOD PROTECTED M_DeferCancel
VAR_INPUT
	i_bDefer : BOOL;
END_VAR
bDeferCancel := i_bDefer;
END_METHOD

METHOD PROTECTED M_FatalError
VAR_INPUT
	i_ErrorMessage : STRING;
END_VAR
M_ResetTimeoutTimer();
M_SetMessage(i_ErrorMessage);
eStep := E_OpStep.IDLE;
q_bError := TRUE;
q_bBusy := FALSE;
bCancel := FALSE;
M_DeferCancel(FALSE);
END_METHOD

METHOD PROTECTED M_Finish
VAR_INPUT
END_VAR
M_ResetTimeoutTimer();
M_SetMessage('Operation finished');
eStep := E_OpStep.IDLE;
q_bBusy := FALSE;
bCancel := FALSE;
M_DeferCancel(FALSE);
END_METHOD

METHOD PUBLIC M_ResetError
VAR_INPUT
END_VAR
q_bError := FALSE;
END_METHOD

METHOD PROTECTED M_ResetTimeoutTimer
VAR_INPUT
END_VAR
fbTimeoutTimer(IN := FALSE);
END_METHOD

METHOD PROTECTED M_RunTimeoutTimer
VAR_INPUT
	i_tTime : TIME; // How long the timer should run before signalling a timeout
END_VAR
fbTimeoutTimer(IN := TRUE, PT := i_tTime);
END_METHOD

METHOD PROTECTED M_SetMessage
VAR_INPUT
	i_sMessage : STRING(EPICS_STRING_SIZE);
END_VAR
iq_sMessageBuffer := i_sMessage;
END_METHOD

METHOD PROTECTED M_TimeoutExpired : BOOL
VAR_INPUT
END_VAR
fbTimeoutTimer(); // Advance timer
M_TimeoutExpired := fbTimeoutTimer.Q;
END_METHOD

END_FUNCTION_BLOCK

// ---- POUs/FB_TransportTube.TcPOU
FUNCTION_BLOCK FB_TransportTube
VAR_INPUT
	i_stConfig : ST_TransportTubeConfig;
	i_bLaserExtIntl : BOOL; // external interlock for laser
END_VAR
VAR_OUTPUT	
	{attribute 'pytmc' := '
		pv: LASER_OK
		io: o
		field: ZNAM LASER_NOT_OK
		field: ONAM LASER_OK
	'}
	q_bLaserOk : BOOL; // Whether the laser is ok for operation
	
	{attribute 'pytmc' := '
		pv:
	'}
	q_stConfig : ST_TransportTubeConfig;
END_VAR
VAR
	bLaserOk : BOOL;
END_VAR

q_stConfig := i_stConfig;
q_bLaserOk := i_bLaserExtIntl AND bLaserOk;

METHOD PUBLIC M_SetLaserOk
VAR_INPUT
	i_bVal : BOOL;
END_VAR
bLaserOk := i_bVal;
END_METHOD

END_FUNCTION_BLOCK

// ---- POUs/Helpers/F_GetTransportTube.TcPOU
FUNCTION F_GetTransportTube : REFERENCE TO FB_TransportTube
VAR_INPUT
	eTT : T_TransportTube;
END_VAR
VAR
END_VAR

CASE eTT OF
E_TransportTube.LS1:
	F_GetTransportTube REF= GVL_TransportTubes.fbLS1;
E_TransportTube.LS5:
	F_GetTransportTube REF= GVL_TransportTubes.fbLS5;
E_TransportTube.LS8:
	F_GetTransportTube REF= GVL_TransportTubes.fbLS8;

E_TransportTube.LD2:
	F_GetTransportTube REF= GVL_TransportTubes.fbLD2;
E_TransportTube.LD4:
	F_GetTransportTube REF= GVL_TransportTubes.fbLD4;
E_TransportTube.LD6:
	F_GetTransportTube REF= GVL_TransportTubes.fbLD6;
E_TransportTube.LD14:
	F_GetTransportTube REF= GVL_TransportTubes.fbLD14;
E_TransportTube.LD10:
	F_GetTransportTube REF= GVL_TransportTubes.fbLD10;
E_TransportTube.LD9:
	F_GetTransportTube REF= GVL_TransportTubes.fbLD9;
E_TransportTube.LD8:
	F_GetTransportTube REF= GVL_TransportTubes.fbLD8;
ELSE // Invalid transport tube
	F_GetTransportTube REF= 0;
END_CASE

END_FUNCTION

// ---- POUs/Operations/FB_VentTransportTube.TcPOU
FUNCTION_BLOCK FB_VentTransportTube EXTENDS FB_TTOperation
VAR_STAT CONSTANT
	(* Expected system states before operation starts*)		
	stExpTTStatus : ST_TransportTubeStatuses := (
		bIonPumpOn:= TRUE,
		bGateValveOpen:= FALSE,
		ePiraniState:= E_PressureState.ValidLo,
		fColdCathodeVal:= 1E-5);
	stTTOp : ST_TransportTubeOps := (
		ePiraniOp := E_GaugeCompOp.STATE,
		eColdCathodeOp := E_GaugeCompOp._LTE
	);
		
	(* Expected system states after operation finishes *)		
	stFinExpTTStatus : ST_TransportTubeStatuses := (
		bIonPumpOn:= FALSE,
		bGateValveOpen:= FALSE,
		eColdCathodeState:= E_PressureState.Off);
	stFinTTOp : ST_TransportTubeOps := (
		ePiraniOp := E_GaugeCompOp.ATM,
		eColdCathodeOp := E_GaugeCompOp.STATE
	);
	
	(* Timeout constants *)
	WAIT_PUMPCART_TIMEOUT : TIME := T#20M;
	VENT_TIMEOUT : TIME := T#20M;
END_VAR

SUPER^(iq_sMessageBuffer := iq_sMessageBuffer);

CASE eStep OF
E_OpStep.IDLE: // Do nothing

E_OpStep.START: // Verify system status
	M_RunTimeoutTimer(STATUS_CHECK_TIMEOUT);
	M_SetMessage('Verifying system status');
	
	IF F_VerifyTransportTubeStatuses(stExpStatus := stExpTTStatus,
		eTransportTube := eTT,
		stStatusOp := stTTOp, 
		bEnforce := TRUE)
	THEN // System status check 
		M_ResetTimeoutTimer();
		M_SetMessage('OPERATOR: Pump inlet port w/ pump cart');
		eStep := E_OpStep.VOT_WAIT_PC;
	END_IF
	
E_OpStep.VOT_WAIT_PC:
	M_RunTimeoutTImer(WAIT_PUMPCART_TIMEOUT);
	
	(* At this point the system must wait for the inlet port of the transport tube to be pumped down by the pump cart. *)
	
	// @TODO. What should this check be???? Need a way to check P-GCC1
	IF FALSE THEN
		M_ResetTimeoutTImer();
		M_SetMessage('Venting');
		eStep := E_OpStep.VOT_VENT;
	END_IF
	
E_OpStep.VOT_VENT:
	M_RunTimeoutTimer(VENT_TIMEOUT);
	fbTT.q_stConfig.stDevices.refIonPump.M_Run(FALSE);
	
	// Vent until atmospheric pressure reached
	IF F_Atm(fbTT.q_stConfig.stDevices.refPiraniGauge.PG.rPRESS) THEN
		M_ResetTimeoutTimer();
		eStep := E_OpStep.VOT_FINISH;
	END_IF
	
E_OpStep.VOT_FINISH:
	IF F_VerifyTransportTubeStatuses(stExpStatus := stFinExpTTStatus,
		eTransportTube := eTT,
		stStatusOp := stFinTTOp, 
		bEnforce := FALSE)
	THEN
		M_Finish();
	ELSE
		M_FatalError('End system status check failed');
	END_IF
	
ELSE
	M_FatalError('Operation is in invalid state');
END_CASE

END_FUNCTION_BLOCK

// ---- POUs/Operations/FB_LaserOn.TcPOU
FUNCTION_BLOCK FB_LaserOn EXTENDS FB_TTOperation
VAR	
	fbPumpSwitchbox : FB_PumpSwitchbox;
	fbPumpTransportTube : FB_PumpTransportTube;
END_VAR
VAR_STAT CONSTANT
	(* Expected system states before operation starts*)		
	stExpPumpStatus : ST_SBPumpStatuses := (
		bRoughingPumpOn:= TRUE, 
		bTurboPumpOn:= FALSE, 
		bIonPumpOn:= TRUE);
	
	stExpValveStatus : ST_SBValveStatuses := (
		bGateValveOpen:= FALSE, 
		bVentValveOpen:= FALSE, 
		bORingPumpValveOpen:= TRUE, 
		bForelineValveOpen:= TRUE, 
		bSlowPumpValveOpen:= FALSE,
		bSBVentOpen:= FALSE,  
		bSBSlowVentOpen:= FALSE);
	
	stExpGaugeReadings : ST_SBGaugeReadings := (
		eDPPiraniState:= E_PressureState.ValidLo,
		fDPColdCathodeVal:= 1E-5,
		ePumpStationPirani1State:= E_PressureState.ValidLo,
		fPumpStationPirani2Val:= 1E-2,
		fPumpStationColdCathodeVal:= 1E-5
	);
	stGaugeReadingsOp : ST_SBGaugeReadingsOp := (
		eDPPiraniOp:= E_GaugeCompOp.STATE, 
		eDPColdCathodeOp:= E_GaugeCompOp._LTE, 
		ePumpStationPirani1Op:= E_GaugeCompOp.STATE, 
		ePumpStationPirani2Op:= E_GaugeCompOp._LTE, 
		ePumpStationColdCathodeOp:= E_GaugeCompOp._LTE);
		
	stExpTTStatus : ST_TransportTubeStatuses := (
		bIonPumpOn:= TRUE,
		bGateValveOpen:= TRUE,
		ePiraniState:= E_PressureState.ValidLo,
		fColdCathodeVal:= 1E-5);
	stTTOp : ST_TransportTubeOps := (
		ePiraniOp := E_GaugeCompOp.STATE,
		eColdCathodeOp := E_GaugeCompOp._LTE
	);
END_VAR

SUPER^(iq_sMessageBuffer := iq_sMessageBuffer);

CASE eStep OF
E_OpStep.IDLE: // Do nothing

E_OpStep.START: // Verify system status	
	M_SetMessage('Verifying system status');

	IF F_Atm(GVL_BTS_VAC.fb_DP_GPI.PG.rPRESS) OR GVL_BTS_VAC.fb_DP_GCC.IG.rPRESS >= 1E-2 THEN
		// Pressure in switchbox too high. Pump down switchbox.
		M_SetMessage('Pumping switchbox');
		eStep := E_OpStep.LTT_RUN_PSB;
		
	ELSIF ABS(GVL_BTS_VAC.fb_DP_GCC.IG.rPRESS - fbTT.q_stConfig.stDevices.refColdCathode.IG.rPRESS) >= 5E-4 THEN
		// Pressure difference between switchbox and transport tube too high
		IF fbTT.q_stConfig.stDevices.refColdCathode.IG.rPRESS > GVL_BTS_VAC.fb_DP_GCC.IG.rPRESS THEN
			M_SetMessage('Pumping transport tube');
			eStep := E_OpStep.LTT_RUN_PTT;
		ELSE			
			M_SetMessage('Pumping switchbox');
			eStep := E_OpStep.LTT_RUN_PSB;
		END_IF 
		
	ELSIF F_VerifySBPumpStatuses(stExpStatus := stExpPumpStatus, bEnforce := FALSE)
	AND F_VerifySBValveStatuses(stExpStatus := stExpValveStatus, bEnforce := FALSE)
	AND F_VerifySBGaugeReadings(stExpReadings := stExpGaugeReadings, stReadingsOp := stGaugeReadingsOp)
	AND F_VerifyTransportTubeStatuses(stExpStatus := stExpTTStatus,
		eTransportTube := eTT,
		stStatusOp := stTTOp, 
		bEnforce := FALSE) 
	THEN 
		// System status check passed
		fbTT.M_SetLaserOk(TRUE);		
	ELSE 
		// System status check failed
		M_FatalError('Failed system status check');
	END_IF
	
E_OpStep.LTT_RUN_PSB: // Pump down switchbox
	M_DeferCancel(TRUE); // Make sure pump switchbox cancels before this operation does
	fbPumpSwitchbox(i_bExecute := TRUE,
		i_bCancel := i_bCancel,
		iq_sMessageBuffer := iq_sMessageBuffer);
		
	IF fbPumpSwitchbox.q_bError THEN
		M_Defercancel(FALSE);
		M_FatalError('Error while pumping switchbox');
	ELSIF NOT fbPumpSwitchbox.q_bBusy THEN
		M_Defercancel(FALSE);
		M_SetMessage('Retrying laser on operation');
		eStep := E_OpStep.START;
	END_IF
	
E_OpStep.LTT_RUN_PTT: // Pump transport tube
	M_DeferCancel(TRUE); // Make sure pump transport tube cancels before this operation does
	fbPumpTransportTube(i_bExecute := TRUE,
		i_bCancel := i_bCancel,
		iq_sMessageBuffer := iq_sMessageBuffer,
		i_eTransportTube := eTT);
		
	IF fbPumpTransportTube.q_bError THEN
		M_Defercancel(FALSE);
		M_FatalError('Error while pumping transport tube');
	ELSIF NOT fbPumpTransportTube.q_bBusy THEN
		M_Defercancel(FALSE);
		M_SetMessage('Retrying laser on operation');
		eStep := E_OpStep.START;
	END_IF
	
ELSE
	M_FatalError('Operation is in invalid state');
END_CASE

END_FUNCTION_BLOCK

// ---- POUs/Operations/FB_PumpSwitchbox.TcPOU
(* Operation for pumping the switchbox *)
FUNCTION_BLOCK FB_PumpSwitchbox EXTENDS FB_Operation
VAR_STAT CONSTANT
	(* Expected system states before operation starts*)
	stExpPumpStatus : ST_SBPumpStatuses := (
		bRoughingPumpOn:= FALSE, 
		bTurboPumpOn:= FALSE, 
		bIonPumpOn:= FALSE);
	
	stExpValveStatus : ST_SBValveStatuses := (
		bGateValveOpen:= FALSE, 
		bVentValveOpen:= FALSE, 
		bORingPumpValveOpen:= FALSE, 
		bForelineValveOpen:= FALSE, 
		bSlowPumpValveOpen:= FALSE,
		bSBVentOpen:= FALSE,  
		bSBSlowVentOpen:= FALSE);
	
	stExpGaugeReadings : ST_SBGaugeReadings := (
		eDPColdCathodeState:= E_PressureState.off,
		ePumpStationColdCathodeState:= E_PressureState.off
	);
	stGaugeReadingsOp : ST_SBGaugeReadingsOp := (
		eDPPiraniOp:= E_GaugeCompOp.ATM, 
		eDPColdCathodeOp:= E_GaugeCompOp.STATE, 
		ePumpStationPirani1Op:= E_GaugeCompOp.ATM, 
		ePumpStationPirani2Op:= E_GaugeCompOp.ATM, 
		ePumpStationColdCathodeOp:= E_GaugeCompOp.STATE);
		
	stExpTTStatus : ST_TransportTubeStatuses := (bGateValveOpen:= FALSE);
	stTTOp : ST_TransportTubeOps := (bIonPumpIgnore:= TRUE);
		
	(* Expected system states after operation finishes *)
	stFinExpPumpStatus : ST_SBPumpStatuses := (
		bRoughingPumpOn:= TRUE, 
		bTurboPumpOn:= FALSE, 
		bIonPumpOn:= TRUE);
	
	stFinExpValveStatus : ST_SBValveStatuses := (
		bGateValveOpen:= FALSE, 
		bVentValveOpen:= FALSE, 
		bORingPumpValveOpen:= TRUE, 
		bForelineValveOpen:= TRUE, 
		bSlowPumpValveOpen:= FALSE,
		bSBVentOpen:= FALSE,  
		bSBSlowVentOpen:= FALSE);
	
	stFinExpGaugeReadings : ST_SBGaugeReadings := (
		eDPPiraniState:= E_PressureState.ValidLo,
		fDPColdCathodeVal := 1E-5,
		ePumpStationPirani1State:= E_PressureState.ValidLo,
		ePumpStationPirani2State:= E_PressureState.ValidLo,
		fPumpStationColdCathodeVal := 1E-5
	);
	stFinGaugeReadingsOp : ST_SBGaugeReadingsOp := (
		eDPPiraniOp:= E_GaugeCompOp.STATE, 
		eDPColdCathodeOp:= E_GaugeCompOp._LTE, 
		ePumpStationPirani1Op:= E_GaugeCompOp.STATE, 
		ePumpStationPirani2Op:= E_GaugeCompOp.STATE, 
		ePumpStationColdCathodeOp:= E_GaugeCompOp._LTE);
		
	stFinExpTTStatus : ST_TransportTubeStatuses := (bGateValveOpen:= FALSE);
	stFinTTOp : ST_TransportTubeOps := (bIonPumpIgnore:= TRUE);
		
	(* Pressure constants *)
	TURBO_READY_PRESS : REAL := 1E-4; // Pressure at which to initiate turbo pump
	ION_READY_PRESS : REAL := 1E-5; // Pressure at which to initiate ion pump
END_VAR

SUPER^(iq_sMessageBuffer := iq_sMessageBuffer);

CASE eStep OF
E_OpStep.IDLE: // Do nothing

E_OpStep.START: // System Status Check
	M_RunTimeoutTimer(STATUS_CHECK_TIMEOUT);
	M_SetMessage('Verifying system status');
	
	IF F_VerifySBPumpStatuses(stExpStatus := stExpPumpStatus, bEnforce := TRUE)
		AND F_VerifySBValveStatuses(stExpStatus := stExpValveStatus, bEnforce := TRUE)
		AND F_VerifySBGaugeReadings(stExpReadings := stExpGaugeReadings, stReadingsOp := stGaugeReadingsOp)
		AND F_VerifyAllTransportTubeStatuses(stExpStatus := stExpTTStatus, 
			stStatusOp := stTTOp, 
			bEnforce := TRUE)
	THEN // System status check passed
		M_ResetTimeoutTimer();
		
		// Make sure pressure difference is low between switchbox and pumping station
		IF ABS(GVL_BTS_VAC.fb_DP_GPI.PG.rPRESS - GVL_BTS_VAC.fb_PP_GPI_1.PG.rPRESS) < 10 THEN
			M_SetMessage('Opening gate valve');
			eStep := E_OpStep.PSB_OPEN_GATE_VALVE;
		ELSE
			M_FatalError('Vent to atmosphere');
		END_IF
	END_IF
	
E_OpStep.PSB_OPEN_GATE_VALVE:  
	M_RunTimeoutTimer(VALVE_TIMEOUT);

	// Open gate valve
	GVL_BTS_VAC.fb_PP_VGC.M_Set_OPN_SW(TRUE);
	
	IF GVL_BTS_VAC.fb_PP_VGC.M_IsOpen() THEN
		M_ResetTimeoutTimer();		
		M_SetMessage('Opening pump station valves');
		eStep := E_OpStep.PSB_OPEN_PUMP_STATION_VALVES;
	END_IF
	
E_OpStep.PSB_OPEN_PUMP_STATION_VALVES:
	M_RunTimeoutTimer(VALVE_TIMEOUT);
	
	// Open pumping station valves
	GVL_BTS_VAC.fb_PP_VRC_1.M_Set_OPN_SW(TRUE);
	GVL_BTS_VAC.fb_PP_VRC_2.M_Set_OPN_SW(TRUE);

	IF GVL_BTS_VAC.fb_PP_VRC_1.iq_stValve.eState = E_ValvePositionState.OPEN AND GVL_BTS_VAC.fb_PP_VRC_2.iq_stValve.eState = E_ValvePositionState.OPEN THEN
		M_ResetTimeoutTimer();
		M_SetMessage('Roughing chamber');
		eStep := E_OpStep.PSB_ROUGH_CHAMBER;
	END_IF
	
E_OpStep.PSB_ROUGH_CHAMBER: // Rough chamber
	M_RunTimeoutTimer(ROUGH_CHAMBER_TIMEOUT);
	
	// Turn on roughing (PMF) pump
	GVL_BTS_VAC.fb_PP_PMF.M_Run(TRUE);

	// Continue roughing until pressure is low enough to start turbo pump
	IF GVL_BTS_VAC.fb_PP_PMF.q_stPump.eState = E_PumpState.pumpRUNNING AND GVL_BTS_VAC.fb_DP_GPI.PG.rPRESS < TURBO_READY_PRESS THEN	
		M_ResetTimeoutTimer();
		M_SetMessage('Turbo pumping chamber');
		eStep := E_OpStep.PSB_TURBO_CHAMBER;
	END_IF
	
E_OpStep.PSB_TURBO_CHAMBER: // Turbo pump down to base pressure
	M_RunTimeoutTimer(TURBO_CHAMBER_TIMEOUT);
	
	// Start Turbo pump
	GVL_BTS_VAC.fb_PP_PTM.M_Run(TRUE);

	// Continue turbo pump until pressure is low enough to start ion pump
	IF GVL_BTS_VAC.fb_PP_PTM.iq_stPTM.eState = E_PumpState.pumpRUNNING AND GVL_BTS_VAC.fb_DP_GCC.IG.rPRESS < ION_READY_PRESS THEN	
		M_ResetTimeoutTimer();
		M_SetMessage('Switching to ion pump');
		eStep := E_OpStep.PSB_SWITCH_TO_ION_PUMP;
	END_IF
	
E_OpStep.PSB_SWITCH_TO_ION_PUMP:
	M_RunTimeoutTimer(PUMP_TIMEOUT);
	
	// Switch to Ion pump
	GVL_BTS_VAC.fb_PP_PIP.M_Run(TRUE);
	
	IF GVL_BTS_VAC.fb_PP_PIP.i_xSP_DI THEN
		M_ResetTimeoutTimer();
		M_SetMessage('Closing gate valve');
		eStep := E_OpStep.PSB_CLOSE_GATE_VALVE;
	END_IF
	
E_OpStep.PSB_CLOSE_GATE_VALVE:
	M_RunTimeoutTimer(VALVE_TIMEOUT);
	
	// Close gate valve
	GVL_BTS_VAC.fb_PP_VGC.M_Set_OPN_SW(FALSE);
	
	IF GVL_BTS_VAC.fb_PP_VGC.M_IsClosed() THEN
		M_ResetTimeoutTimer();
		M_SetMessage('Stopping turbo pump');
		eStep := E_OpStep.PSB_STOP_TURBO_PUMP;
	END_IF
	
E_OpStep.PSB_STOP_TURBO_PUMP:
	M_RunTimeoutTimer(PUMP_TIMEOUT);
	
	// Turn off turbo pump
	GVL_BTS_VAC.fb_PP_PTM.M_Run(FALSE);
	
	IF GVL_BTS_VAC.fb_PP_PTM.iq_stPTM.eState = E_PumpState.pumpSTOPPED THEN
		M_ResetTimeoutTimer();
		eStep := E_OpStep.PSB_FINISH;
	END_IF
	
E_OpStep.PSB_FINISH: // System Status Check
	IF F_VerifySBPumpStatuses(stExpStatus := stFinExpPumpStatus, bEnforce := FALSE)
		AND F_VerifySBValveStatuses(stExpStatus := stFinExpValveStatus, bEnforce := FALSE)
		AND F_VerifySBGaugeReadings(stExpReadings := stFinExpGaugeReadings, stReadingsOp := stFinGaugeReadingsOp)
		AND F_VerifyAllTransportTubeStatuses(stExpStatus := stFinExpTTStatus, 
			stStatusOp := stFinTTOp, 
			bEnforce := FALSE)
	THEN
		M_Finish();
	ELSE
		M_FatalError('End system status check failed');
	END_IF
	
ELSE
	M_FatalError('Operation is in invalid state');
END_CASE

END_FUNCTION_BLOCK

// ---- POUs/SystemStatusChecks/Switchbox/F_VerifySBPumpStatuses.TcPOU
(* Verify that the statuses of the switchbox pumps match the expected statuses *)
FUNCTION F_VerifySBPumpStatuses : BOOL
VAR_INPUT
	stExpStatus : ST_SBPumpStatuses; // The expected state of the system
	bEnforce : BOOL; // Whether to try forcing the states
END_VAR
VAR
	stStatus : ST_SBPumpStatuses;
END_VAR

stStatus := F_GetSBPumpStatuses();

IF bEnforce THEN
	// Try setting system states to the expected states
	F_SetSBPumpStatuses(stExpStatus);
END_IF

// Return true if the expected status matches the actual status
F_VerifySBPumpStatuses := stExpStatus.bRoughingPumpOn = stStatus.bRoughingPumpOn
	AND stExpStatus.bTurboPumpOn = stStatus.bTurboPumpOn
	AND stExpStatus.bIonPumpOn = stStatus.bIonPumpOn;

END_FUNCTION

// ---- POUs/SystemStatusChecks/Switchbox/F_GetSBPumpStatuses.TcPOU
(* Get the status of the pumps for the switchbox *)
FUNCTION F_GetSBPumpStatuses : ST_SBPumpStatuses
VAR_INPUT
END_VAR
VAR
	stStatus : ST_SBPumpStatuses := (
		bRoughingPumpOn:= GVL_BTS_VAC.fb_PP_PMF.q_stPump.i_xIsRun,
		bTurboPumpOn:= GVL_BTS_VAC.fb_PP_PTM.q_RunDO, 
		bIonPumpOn:= GVL_BTS_VAC.fb_PP_PIP.q_xHVEna_DO);
END_VAR

F_GetSBPumpStatuses := stStatus;

END_FUNCTION

// ---- POUs/SystemStatusChecks/Switchbox/F_SetSBPumpStatuses.TcPOU
FUNCTION F_SetSBPumpStatuses : BOOL
VAR_INPUT
	stExpStatus : ST_SBPumpStatuses;
END_VAR
VAR
END_VAR

GVL_BTS_VAC.fb_PP_PMF.M_Run(stExpStatus.bRoughingPumpOn); 
GVL_BTS_VAC.fb_PP_PTM.M_Run(stExpStatus.bTurboPumpOn);
GVL_BTS_VAC.fb_PP_PIP.M_Run(stExpStatus.bIonPumpOn);

END_FUNCTION

// ---- POUs/SystemStatusChecks/Switchbox/F_VerifySBGaugeReadings.TcPOU
FUNCTION F_VerifySBGaugeReadings : BOOL
VAR_INPUT
	stExpReadings : ST_SBGaugeReadings;
	stReadingsOp : ST_SBGaugeReadingsOp;
END_VAR
VAR
	stStatus : ST_SBGaugeReadings;
END_VAR

stStatus := F_GetSBGaugeReadings();

// Return true if the expected status matches the actual status
F_VerifySBGaugeReadings := 
	F_CompareGauge(
		eCompOp := stReadingsOp.eDPColdCathodeOp,
		fReading := stStatus.fDPColdCathodeVal,
		eState := stStatus.eDPColdCathodeState,
		fExpReading := stExpReadings.fDPColdCathodeVal,
		eExpState := stExpReadings.eDPColdCathodeState) 
	AND F_CompareGauge(
		eCompOp := stReadingsOp.eDPPiraniOp,
		fReading := stStatus.fDPPiraniVal,
		eState := stStatus.eDPPiraniState,
		fExpReading := stExpReadings.fDPPiraniVal,
		eExpState := stExpReadings.eDPPiraniState)
	AND F_CompareGauge(
		eCompOp := stReadingsOp.ePumpStationColdCathodeOp,
		fReading := stStatus.fPumpStationColdCathodeVal,
		eState := stStatus.ePumpStationColdCathodeState,
		fExpReading := stExpReadings.fPumpStationColdCathodeVal,
		eExpState := stExpReadings.ePumpStationColdCathodeState)
	AND F_CompareGauge(
		eCompOp := stReadingsOp.ePumpStationPirani1Op,
		fReading := stStatus.fPumpStationPirani1Val,
		eState := stStatus.ePumpStationPirani1State,
		fExpReading := stExpReadings.fPumpStationPirani1Val,
		eExpState := stExpReadings.ePumpStationPirani1State)
	AND F_CompareGauge(
		eCompOp := stReadingsOp.ePumpStationPirani2Op,
		fReading := stStatus.fPumpStationPirani2Val,
		eState := stStatus.ePumpStationPirani2State,
		fExpReading := stExpReadings.fPumpStationPirani2Val,
		eExpState := stExpReadings.ePumpStationPirani2State);

END_FUNCTION

// ---- POUs/SystemStatusChecks/Switchbox/F_GetSBGaugeReadings.TcPOU
FUNCTION F_GetSBGaugeReadings : ST_SBGaugeReadings
VAR_INPUT
END_VAR
VAR
	stReadings : ST_SBGaugeReadings := (
		fDPPiraniVal:= GVL_BTS_VAC.fb_DP_GPI.PG.rPRESS,
		eDPPiraniState:= GVL_BTS_VAC.fb_DP_GPI.PG.eState,
		fDPColdCathodeVal:= GVL_BTS_VAC.fb_DP_GCC.IG.rPRESS,
		eDPColdCathodeState:= GVL_BTS_VAC.fb_DP_GCC.IG.eState,
		fPumpStationPirani1Val:= GVL_BTS_VAC.fb_PP_GPI_1.PG.rPRESS,
		ePumpStationPirani1State:= GVL_BTS_VAC.fb_PP_GPI_1.PG.eState,
		fPumpStationPirani2Val:= GVL_BTS_VAC.fb_PP_GPI_2.PG.rPRESS, 
		ePumpStationPirani2State:= GVL_BTS_VAC.fb_PP_GPI_2.PG.eState,
		fPumpStationColdCathodeVal:= GVL_BTS_VAC.fb_PP_GCC.IG.rPRESS,
		ePumpStationColdCathodeState:= GVL_BTS_VAC.fb_PP_GCC.IG.eState);
END_VAR

F_GetSBGaugeReadings := stReadings;

END_FUNCTION

// ---- POUs/SystemStatusChecks/TransportTubes/F_VerifyAllTransportTubeStatuses.TcPOU
FUNCTION F_VerifyAllTransportTubeStatuses : BOOL
VAR_INPUT
	stExpStatus : ST_TransportTubeStatuses;
	stStatusOp : ST_TransportTubeOps;
	bEnforce : BOOL;
END_VAR
VAR
	nIter : UINT;
	bResult : BOOL := TRUE;
END_VAR

FOR nIter := 1 TO GVL_TransportTubes.NUM_TRANSPORT_TUBES DO
	bResult := bResult AND F_VerifyTransportTubeStatuses(
		stExpStatus := stExpStatus,
		stStatusOp := stStatusOp,
		eTransportTube := GVL_TransportTubes.aTubes[nIter],
		bEnforce := bEnforce);
END_FOR

F_VerifyAllTransportTubeStatuses := bResult;

END_FUNCTION

// ---- POUs/Operations/FB_SlowPumpSwitchbox.TcPOU
(* Operation for pumping the switchbox *)
FUNCTION_BLOCK FB_SlowPumpSwitchbox EXTENDS FB_Operation
VAR_STAT CONSTANT
	(* Expected system states before operation starts*)
	stExpPumpStatus : ST_SBPumpStatuses := (
		bRoughingPumpOn:= FALSE, 
		bTurboPumpOn:= FALSE, 
		bIonPumpOn:= FALSE);
	
	stExpValveStatus : ST_SBValveStatuses := (
		bGateValveOpen:= FALSE, 
		bVentValveOpen:= FALSE, 
		bORingPumpValveOpen:= FALSE, 
		bForelineValveOpen:= FALSE, 
		bSlowPumpValveOpen:= FALSE,
		bSBVentOpen:= FALSE,  
		bSBSlowVentOpen:= FALSE);
	
	stExpGaugeReadings : ST_SBGaugeReadings := (
		eDPColdCathodeState:= E_PressureState.off,
		ePumpStationColdCathodeState:= E_PressureState.off
	);
	stGaugeReadingsOp : ST_SBGaugeReadingsOp := (
		eDPPiraniOp:= E_GaugeCompOp.ATM, 
		eDPColdCathodeOp:= E_GaugeCompOp.STATE, 
		ePumpStationPirani1Op:= E_GaugeCompOp.ATM, 
		ePumpStationPirani2Op:= E_GaugeCompOp.ATM, 
		ePumpStationColdCathodeOp:= E_GaugeCompOp.STATE);
		
	stExpTTStatus : ST_TransportTubeStatuses := (bGateValveOpen:= FALSE);
	stTTOp : ST_TransportTubeOps := (bIonPumpIgnore:= TRUE);
		
	(* Expected system states after operation finishes *)
	stFinExpPumpStatus : ST_SBPumpStatuses := (
		bRoughingPumpOn:= TRUE, 
		bTurboPumpOn:= FALSE, 
		bIonPumpOn:= TRUE);
	
	stFinExpValveStatus : ST_SBValveStatuses := (
		bGateValveOpen:= FALSE, 
		bVentValveOpen:= FALSE, 
		bORingPumpValveOpen:= TRUE, 
		bForelineValveOpen:= TRUE, 
		bSlowPumpValveOpen:= FALSE,
		bSBVentOpen:= FALSE,  
		bSBSlowVentOpen:= FALSE);
	
	stFinExpGaugeReadings : ST_SBGaugeReadings := (
		eDPPiraniState:= E_PressureState.ValidLo,
		fDPColdCathodeVal := 1E-5,
		ePumpStationPirani1State:= E_PressureState.ValidLo,
		ePumpStationPirani2State:= E_PressureState.ValidLo,
		fPumpStationColdCathodeVal := 1E-5
	);
	stFinGaugeReadingsOp : ST_SBGaugeReadingsOp := (
		eDPPiraniOp:= E_GaugeCompOp.STATE, 
		eDPColdCathodeOp:= E_GaugeCompOp._LTE, 
		ePumpStationPirani1Op:= E_GaugeCompOp.STATE, 
		ePumpStationPirani2Op:= E_GaugeCompOp.STATE, 
		ePumpStationColdCathodeOp:= E_GaugeCompOp._LTE);
		
	stFinExpTTStatus : ST_TransportTubeStatuses := (bGateValveOpen:= FALSE);
	stFinTTOp : ST_TransportTubeOps := (bIonPumpIgnore:= TRUE);
		
	(* Pressure constants *)
	TURBO_READY_PRESS : REAL := 1E-4; // Pressure at which to initiate turbo pump
	ION_READY_PRESS : REAL := 1E-5; // Pressure at which to initiate ion pump
END_VAR

SUPER^(iq_sMessageBuffer := iq_sMessageBuffer);

CASE eStep OF
E_OpStep.IDLE: // Do nothing

E_OpStep.START: // System Status Check
	M_RunTimeoutTimer(STATUS_CHECK_TIMEOUT);
	M_SetMessage('Verifying system status');
	
	IF F_VerifySBPumpStatuses(stExpStatus := stExpPumpStatus, bEnforce := TRUE)
		AND F_VerifySBValveStatuses(stExpStatus := stExpValveStatus, bEnforce := TRUE)
		AND F_VerifySBGaugeReadings(stExpReadings := stExpGaugeReadings, stReadingsOp := stGaugeReadingsOp)
		AND F_VerifyAllTransportTubeStatuses(stExpStatus := stExpTTStatus, 
			stStatusOp := stTTOp, 
			bEnforce := TRUE)
	THEN // System status check passed
		M_ResetTimeoutTimer();
		
		// Make sure pressure difference is low between switchbox and pumping station
		IF ABS(GVL_BTS_VAC.fb_DP_GPI.PG.rPRESS - GVL_BTS_VAC.fb_PP_GPI_1.PG.rPRESS) < 10 THEN
			M_SetMessage('Opening gate valve');
			eStep := E_OpStep.SPSB_OPEN_GATE_VALVE;
		ELSE
			M_FatalError('Vent to atmosphere');
		END_IF
	END_IF
	
E_OpStep.SPSB_OPEN_GATE_VALVE:  
	M_RunTimeoutTimer(VALVE_TIMEOUT);

	// Open gate valve
	GVL_BTS_VAC.fb_PP_VGC.M_Set_OPN_SW(TRUE);
	
	IF GVL_BTS_VAC.fb_PP_VGC.M_IsOpen() THEN
		M_ResetTimeoutTimer();		
		M_SetMessage('Opening pump station valves');
		eStep := E_OpStep.SPSB_OPEN_PUMP_STATION_VALVES;
	END_IF
	
E_OpStep.SPSB_OPEN_PUMP_STATION_VALVES:
	M_RunTimeoutTimer(VALVE_TIMEOUT);
	
	// Open pumping station valves
	GVL_BTS_VAC.fb_PP_VRC_1.M_Set_OPN_SW(TRUE);
	GVL_BTS_VAC.fb_PP_VRC_3.M_Set_OPN_SW(TRUE);

	IF GVL_BTS_VAC.fb_PP_VRC_1.iq_stValve.eState = E_ValvePositionState.OPEN AND GVL_BTS_VAC.fb_PP_VRC_3.iq_stValve.eState = E_ValvePositionState.OPEN THEN
		M_ResetTimeoutTimer();
		M_SetMessage('Roughing chamber');
		eStep := E_OpStep.SPSB_ROUGH_CHAMBER;
	END_IF
	
E_OpStep.SPSB_ROUGH_CHAMBER: // Rough chamber
	M_RunTimeoutTimer(ROUGH_CHAMBER_TIMEOUT);
	
	// Turn on roughing (PMF) pump
	GVL_BTS_VAC.fb_PP_PMF.M_Run(TRUE);

	// Continue roughing until pressure is low enough to start turbo pump
	IF GVL_BTS_VAC.fb_PP_PMF.q_stPump.eState = E_PumpState.pumpRUNNING AND GVL_BTS_VAC.fb_DP_GPI.PG.rPRESS < TURBO_READY_PRESS THEN	
		M_ResetTimeoutTimer();
		M_SetMessage('Opening foreline valve');
		eStep := E_OpStep.SPSB_OPEN_FORELINE_VALVE;
	END_IF
	
E_OpStep.SPSB_OPEN_FORELINE_VALVE:
	M_RunTimeoutTimer(VALVE_TIMEOUT);
	
	// Open foreline valve
	GVL_BTS_VAC.fb_PP_VRC_2.M_Set_OPN_SW(TRUE);
	
	IF GVL_BTS_VAC.fb_PP_VRC_2.iq_stValve.eState = E_ValvePositionState.OPEN THEN
		M_ResetTimeoutTImer();
		M_SetMessage('Turbo pumping chamber');
		eStep := E_OpStep.SPSB_TURBO_CHAMBER;
	END_IF
	
E_OpStep.SPSB_TURBO_CHAMBER: // Turbo pump down to base pressure
	M_RunTimeoutTimer(TURBO_CHAMBER_TIMEOUT);
	
	// Start Turbo pump
	GVL_BTS_VAC.fb_PP_PTM.M_Run(TRUE);

	// Continue turbo pump until pressure is low enough to start ion pump
	IF GVL_BTS_VAC.fb_PP_PTM.iq_stPTM.eState = E_PumpState.pumpRUNNING AND GVL_BTS_VAC.fb_DP_GCC.IG.rPRESS < ION_READY_PRESS THEN	
		M_ResetTimeoutTimer();
		M_SetMessage('Switching to ion pump');
		eStep := E_OpStep.SPSB_SWITCH_TO_ION_PUMP;
	END_IF
	
E_OpStep.SPSB_SWITCH_TO_ION_PUMP:
	M_RunTimeoutTimer(PUMP_TIMEOUT);
	
	// Switch to Ion pump
	GVL_BTS_VAC.fb_PP_PIP.M_Run(TRUE);
	
	IF GVL_BTS_VAC.fb_PP_PIP.i_xSP_DI THEN
		M_ResetTimeoutTimer();
		M_SetMessage('Closing valves');
		eStep := E_OpStep.SPSB_CLOSE_VALVES;
	END_IF
	
E_OpStep.SPSB_CLOSE_VALVES:
	M_RunTimeoutTimer(VALVE_TIMEOUT);
	
	// Close gate valve
	GVL_BTS_VAC.fb_PP_VGC.M_Set_OPN_SW(FALSE);
	GVL_BTS_VAC.fb_PP_VRC_3.M_Set_OPN_SW(FALSE);
	
	IF GVL_BTS_VAC.fb_PP_VGC.M_IsClosed() AND GVL_BTS_VAC.fb_PP_VRC_3.iq_stValve.eState = E_ValvePositionState.CLOSED THEN
		M_ResetTimeoutTimer();
		M_SetMessage('Stopping turbo pump');
		eStep := E_OpStep.SPSB_STOP_TURBO_PUMP;
	END_IF
	
E_OpStep.SPSB_STOP_TURBO_PUMP:
	M_RunTimeoutTimer(PUMP_TIMEOUT);
	
	// Turn off turbo pump
	GVL_BTS_VAC.fb_PP_PTM.M_Run(FALSE);
	
	IF GVL_BTS_VAC.fb_PP_PTM.iq_stPTM.eState = E_PumpState.pumpSTOPPED THEN
		M_ResetTimeoutTimer();
		eStep := E_OpStep.SPSB_FINISH;
	END_IF
	
E_OpStep.SPSB_FINISH: // System Status Check
	IF F_VerifySBPumpStatuses(stExpStatus := stFinExpPumpStatus, bEnforce := FALSE)
		AND F_VerifySBValveStatuses(stExpStatus := stFinExpValveStatus, bEnforce := FALSE)
		AND F_VerifySBGaugeReadings(stExpReadings := stFinExpGaugeReadings, stReadingsOp := stFinGaugeReadingsOp)
		AND F_VerifyAllTransportTubeStatuses(stExpStatus := stFinExpTTStatus, 
			stStatusOp := stFinTTOp, 
			bEnforce := FALSE)
	THEN
		M_Finish();
	ELSE
		M_FatalError('End system status check failed');
	END_IF
	
ELSE
	M_FatalError('Operation is in invalid state');
END_CASE

END_FUNCTION_BLOCK

// ---- POUs/Operations/FB_VentPumpStation.TcPOU
(* Operation for venting the pumping station *)
FUNCTION_BLOCK FB_VentPumpStation EXTENDS FB_Operation
VAR_INPUT
END_VAR
VAR_OUTPUT
END_VAR
VAR_STAT CONSTANT
	(* Expected system states before operation starts*)
	stExpPumpStatus : ST_SBPumpStatuses := (
		bRoughingPumpOn:= TRUE, 
		bTurboPumpOn:= FALSE, 
		bIonPumpOn:= FALSE);
	
	stExpValveStatus : ST_SBValveStatuses := (
		bGateValveOpen:= FALSE, 
		bVentValveOpen:= FALSE, 
		bORingPumpValveOpen:= TRUE, 
		bForelineValveOpen:= TRUE,
		bSlowPumpValveOpen:= FALSE,
		bSBVentOpen:= FALSE,  
		bSBSlowVentOpen:= FALSE);
	
	stExpGaugeReadings : ST_SBGaugeReadings := (
		eDPColdCathodeState:= E_PressureState.Off,
		ePumpStationPirani1State:= E_PressureState.ValidLo,
		fPumpStationColdCathodeVal:= 1E-5
	);
	stGaugeReadingsOp : ST_SBGaugeReadingsOp := (
		eDPPiraniOp:= E_GaugeCompOp.ATM, 
		eDPColdCathodeOp:= E_GaugeCompOp.STATE, 
		ePumpStationPirani1Op:= E_GaugeCompOp.STATE, 
		ePumpStationPirani2Op:= E_GaugeCompOp.IGNORE, 
		ePumpStationColdCathodeOp:= E_GaugeCompOp._LTE);
			
	stExpTTStatus : ST_TransportTubeStatuses := (bGateValveOpen:= FALSE);
	stTTOp : ST_TransportTubeOps := (bIonPumpIgnore:= TRUE);
		
	(* Expected system states after operation finishes *)
	stFinExpPumpStatus : ST_SBPumpStatuses := (
		bRoughingPumpOn:= FALSE, 
		bTurboPumpOn:= FALSE, 
		bIonPumpOn:= FALSE);
	
	stFinExpValveStatus : ST_SBValveStatuses := (
		bGateValveOpen:= FALSE, 
		bVentValveOpen:= FALSE, 
		bORingPumpValveOpen:= TRUE, 
		bForelineValveOpen:= TRUE, 
		bSlowPumpValveOpen:= FALSE,
		bSBVentOpen:= FALSE,  
		bSBSlowVentOpen:= FALSE);
	
	stFinExpGaugeReadings : ST_SBGaugeReadings := (
		eDPColdCathodeState := E_PressureState.Off,
		ePumpStationColdCathodeState := E_PressureState.Off
	);
	stFinGaugeReadingsOp : ST_SBGaugeReadingsOp := (
		eDPPiraniOp:= E_GaugeCompOp.ATM, 
		eDPColdCathodeOp:= E_GaugeCompOp.STATE, 
		ePumpStationPirani1Op:= E_GaugeCompOp.ATM, 
		ePumpStationPirani2Op:= E_GaugeCompOp.ATM, 
		ePumpStationColdCathodeOp:= E_GaugeCompOp.STATE);
		
	stFinExpTTStatus : ST_TransportTubeStatuses := (bGateValveOpen:= FALSE);
	stFinTTOp : ST_TransportTubeOps := (bIonPumpIgnore:= TRUE);

	(* Timeout constants *)
	VENT_TIMEOUT : TIME := T#20S;
END_VAR

SUPER^(iq_sMessageBuffer := iq_sMessageBuffer);

CASE eStep OF
E_OpStep.IDLE: // Do nothing

E_OpStep.START: // System Status Check
	M_RunTimeoutTimer(STATUS_CHECK_TIMEOUT);
	M_SetMessage('Verifying system status');
	
	IF F_VerifySBPumpStatuses(stExpStatus := stExpPumpStatus, bEnforce := TRUE)
		AND F_VerifySBValveStatuses(stExpStatus := stExpValveStatus, bEnforce := TRUE)
		AND F_VerifySBGaugeReadings(stExpReadings := stExpGaugeReadings, stReadingsOp := stGaugeReadingsOp)
		AND F_VerifyAllTransportTubeStatuses(stExpStatus := stExpTTStatus, 
			stStatusOp := stTTOp, 
			bEnforce := TRUE)
	THEN // System status check passed
		M_ResetTimeoutTimer();
		M_SetMessage('Venting');
		eStep := E_OpStep.VPS_VENT;
	END_IF
	
E_OpStep.VPS_VENT: // Vent pump station to atmospheric pressure
	M_RunTimeoutTimer(VENT_TIMEOUT);

	// Redundant equipment safety checks
	GVL_BTS_VAC.fb_PP_PTM.M_Run(FALSE);
	GVL_BTS_VAC.fb_PP_PMF.M_Run(FALSE);
	IF GVL_BTS_VAC.fb_PP_VGC.M_IsClosed() THEN		
		// Open pump station vent
		GVL_BTS_VAC.fb_PP_VVC.M_Open(TRUE);
		
		// Vent until atmoshperic pressure reached
		IF F_Atm(GVL_BTS_VAC.fb_PP_GPI_1.PG.rPRESS) THEN
			M_ResetTimeoutTimer();
			M_SetMessage('Venting finished. Closing vent');
			eStep := E_OpStep.VPS_CLOSE_VENT;
		END_IF
	ELSE
		M_FatalError('Gate valve is open');
	END_IF
	
E_OpStep.VPS_CLOSE_VENT:
	M_RunTimeoutTimer(VALVE_TIMEOUT);

	// Close vent
	GVL_BTS_VAC.fb_PP_VVC.M_Open(FALSE);
	
	IF GVL_BTS_VAC.fb_PP_VVC.M_IsClosed() THEN
		M_ResetTimeoutTimer();
		eStep := E_OpStep.VPS_FINISH;
	END_IF
	
E_OpStep.VPS_FINISH: // System status check
	IF F_VerifySBPumpStatuses(stExpStatus := stFinExpPumpStatus, bEnforce := FALSE)
	AND F_VerifySBValveStatuses(stExpStatus := stFinExpValveStatus, bEnforce := FALSE)
	AND F_VerifySBGaugeReadings(stExpReadings := stFinExpGaugeReadings, stReadingsOp := stFinGaugeReadingsOp)
	AND F_VerifyAllTransportTubeStatuses(stExpStatus := stFinExpTTStatus, 
		stStatusOp := stFinTTOp,
		bEnforce := FALSE)
	THEN
		M_Finish();
	ELSE
		M_FatalError('End system status check failed');
	END_IF
	
ELSE
	M_FatalError('Operation is in invalid state');
END_CASE

END_FUNCTION_BLOCK

// ---- POUs/Operations/FB_VentSwitchbox.TcPOU
(* Operation for venting the switchbox *)
FUNCTION_BLOCK FB_VentSwitchbox EXTENDS FB_Operation
VAR_STAT CONSTANT
	(* Expected system states before operation starts*)
	stExpPumpStatus : ST_SBPumpStatuses := (
		bRoughingPumpOn:= TRUE, 
		bTurboPumpOn:= FALSE, 
		bIonPumpOn:= TRUE);
	
	stExpValveStatus : ST_SBValveStatuses := (
		bGateValveOpen:= TRUE, 
		bVentValveOpen:= FALSE, 
		bORingPumpValveOpen:= TRUE, 
		bForelineValveOpen:= TRUE,
		bSlowPumpValveOpen:= FALSE,
		bSBVentOpen:= FALSE,  
		bSBSlowVentOpen:= FALSE);
	
	stExpGaugeReadings : ST_SBGaugeReadings := (
		eDPPiraniState:= E_PressureState.ValidLo,
		fDPColdCathodeVal:= 1E-5,
		ePumpStationPirani1State:= E_PressureState.ValidLo,
		ePumpStationPirani2State:= E_PressureState.ValidLo,
		fPumpStationColdCathodeVal:= 1E-5
	);
	stGaugeReadingsOp : ST_SBGaugeReadingsOp := (
		eDPPiraniOp:= E_GaugeCompOp.STATE, 
		eDPColdCathodeOp:= E_GaugeCompOp._LTE, 
		ePumpStationPirani1Op:= E_GaugeCompOp.STATE, 
		ePumpStationPirani2Op:= E_GaugeCompOp.STATE, 
		ePumpStationColdCathodeOp:= E_GaugeCompOp._LTE);
		
	stExpTTStatus : ST_TransportTubeStatuses := (bGateValveOpen:= FALSE);
	stTTOp : ST_TransportTubeOps := (bIonPumpIgnore:= TRUE);
		
	(* Expected system states after operation finishes *)
	stFinExpPumpStatus : ST_SBPumpStatuses := (
		bRoughingPumpOn:= FALSE, 
		bTurboPumpOn:= FALSE, 
		bIonPumpOn:= FALSE);
	
	stFinExpValveStatus : ST_SBValveStatuses := (
		bGateValveOpen:= FALSE, 
		bVentValveOpen:= FALSE, 
		bORingPumpValveOpen:= FALSE, 
		bForelineValveOpen:= FALSE, 
		bSlowPumpValveOpen:= FALSE,
		bSBVentOpen:= FALSE,  
		bSBSlowVentOpen:= FALSE);
	
	stFinExpGaugeReadings : ST_SBGaugeReadings := (
		eDPColdCathodeState := E_PressureState.Off,
		ePumpStationColdCathodeState := E_PressureState.Off
	);
	stFinGaugeReadingsOp : ST_SBGaugeReadingsOp := (
		eDPPiraniOp:= E_GaugeCompOp.ATM, 
		eDPColdCathodeOp:= E_GaugeCompOp.STATE, 
		ePumpStationPirani1Op:= E_GaugeCompOp.ATM, 
		ePumpStationPirani2Op:= E_GaugeCompOp.ATM, 
		ePumpStationColdCathodeOp:= E_GaugeCompOp.STATE);
		
	stFinExpTTStatus : ST_TransportTubeStatuses := (bGateValveOpen:= FALSE);
	stFinTTOp : ST_TransportTubeOps := (bIonPumpIgnore:= TRUE);
		
	(* Timeout constants *)
	VENT_TIMEOUT : TIME := T#20M;
END_VAR

SUPER^(iq_sMessageBuffer := iq_sMessageBuffer);

CASE eStep OF
E_OpStep.IDLE: // Do nothing

E_OpStep.START: // Verify system status
	M_RunTimeoutTimer(STATUS_CHECK_TIMEOUT);
	M_SetMessage('Verifying system status');
	
	IF F_VerifySBPumpStatuses(stExpStatus := stExpPumpStatus, bEnforce := TRUE)
		AND F_VerifySBValveStatuses(stExpStatus := stExpValveStatus, bEnforce := TRUE)
		AND F_VerifySBGaugeReadings(stExpReadings := stExpGaugeReadings, stReadingsOp := stGaugeReadingsOp)
		AND F_VerifyAllTransportTubeStatuses(stExpStatus := stExpTTStatus, 
			stStatusOp := stTTOp,
			bEnforce := TRUE)
	THEN // System status check 
		M_ResetTimeoutTimer();
		M_SetMessage('Closing gate valve');
		eStep := E_OpStep.VSB_CLOSE_GATE_VALVE;
	END_IF
	
E_OpStep.VSB_CLOSE_GATE_VALVE:
	M_RunTimeoutTimer(VALVE_TIMEOUT);
	
	// Close gate valve to pump station to isolate pumps
	GVL_BTS_VAC.fb_PP_VGC.M_Set_OPN_SW(FALSE);
	
	IF GVL_BTS_VAC.fb_PP_VGC.M_IsClosed() THEN
		M_ResetTimeoutTimer();
		M_SetMessage('Closing foreline valve');
		eStep := E_OpStep.VSB_CLOSE_FORELINE_VALVE;
	END_IF
	
E_OpStep.VSB_CLOSE_FORELINE_VALVE:
	M_RunTimeoutTimer(VALVE_TIMEOUT);
	
	// Close valves to pumping station to isolate pumps
	GVL_BTS_VAC.fb_PP_VRC_2.M_Set_OPN_SW(FALSE);
	
	IF GVL_BTS_VAC.fb_PP_VRC_2.iq_stValve.eState = E_ValvePositionState.CLOSED THEN
		M_ResetTimeoutTimer();
		M_SetMessage('Turning off roughing and ion pump');
		eStep := E_OpStep.VSB_TURN_OFF_PUMPS;
	END_IF
	
E_OpStep.VSB_TURN_OFF_PUMPS:
	M_RunTimeoutTimer(PUMP_TIMEOUT);
	
	// Turn off pumping station pumps
	GVL_BTS_VAC.fb_PP_PMF.M_Run(FALSE);
	GVL_BTS_VAC.fb_PP_PIP.M_Run(FALSE);
	
	IF GVL_BTS_VAC.fb_PP_PMF.q_stPump.eState = E_PumpState.pumpSTOPPED AND NOT GVL_BTS_VAC.fb_PP_PIP.stPump.i_xSP_DI THEN
		M_ResetTimeoutTimer();
		M_SetMessage('Closing O-Ring valve');
		eStep := E_OpStep.VSB_CLOSE_ORING_VALVE;
	END_IF
	
E_OpStep.VSB_CLOSE_ORING_VALVE:
	M_RunTimeoutTimer(VALVE_TIMEOUT);
	
	// Close O-Ring pump valve
	GVL_BTS_VAC.fb_PP_VRC_1.M_Set_OPN_SW(FALSE);

	IF GVL_BTS_VAC.fb_PP_VRC_1.iq_stValve.eState = E_ValvePositionState.CLOSED THEN
		M_ResetTimeoutTimer();
		M_SetMessage('Venting');
		eStep := E_OpStep.VSB_VENT;
	END_IF
	
E_OpStep.VSB_VENT:
	M_RunTimeoutTimer(VENT_TIMEOUT);
		
	// Open switchbox vent
	GVL_BTS_VAC.fb_VP_VVC_1.M_Close(FALSE);
	
	// Vent until atmospheric pressure reached in the switchbox
	IF F_Atm(GVL_BTS_VAC.fb_DP_GPI.PG.rPRESS) THEN
		M_ResetTimeoutTimer();
		eStep := E_OpStep.VSB_CLOSE_VENT;
	END_IF
	

E_OpStep.VSB_CLOSE_VENT:
	GVL_BTS_VAC.fb_VP_VVC_1.M_Close(TRUE);
	// How to verfiy the vent is closed?
	eStep := E_OpStep.VSB_FINISH;
	
E_OpStep.VSB_FINISH:
	IF F_VerifySBPumpStatuses(stExpStatus := stFinExpPumpStatus, bEnforce := FALSE)
		AND F_VerifySBValveStatuses(stExpStatus := stFinExpValveStatus, bEnforce := FALSE)
		AND F_VerifySBGaugeReadings(stExpReadings := stFinExpGaugeReadings, stReadingsOp := stFinGaugeReadingsOp)
		AND F_VerifyAllTransportTubeStatuses(stExpStatus := stFinExpTTStatus, 
			stStatusOp := stFinTTOp,
			bEnforce := FALSE)
	THEN
		M_Finish();
	ELSE
		M_FatalError('End system status check failed');
	END_IF
	
ELSE
	M_FatalError('Operation is in invalid state');
END_CASE

END_FUNCTION_BLOCK

// ---- POUs/Operations/FB_SlowVentSwitchbox.TcPOU
(* Operation for venting the switchbox *)
FUNCTION_BLOCK FB_SlowVentSwitchbox EXTENDS FB_Operation
VAR_INPUT
END_VAR
VAR_OUTPUT
END_VAR
VAR_STAT CONSTANT
	(* Expected system states before operation starts*)
	stExpPumpStatus : ST_SBPumpStatuses := (
		bRoughingPumpOn:= TRUE, 
		bTurboPumpOn:= FALSE, 
		bIonPumpOn:= TRUE);
	
	stExpValveStatus : ST_SBValveStatuses := (
		bGateValveOpen:= TRUE, 
		bVentValveOpen:= FALSE, 
		bORingPumpValveOpen:= TRUE, 
		bForelineValveOpen:= TRUE,
		bSlowPumpValveOpen:= FALSE,
		bSBVentOpen:= FALSE,  
		bSBSlowVentOpen:= FALSE);
	
	stExpGaugeReadings : ST_SBGaugeReadings := (
		eDPPiraniState:= E_PressureState.ValidLo,
		fDPColdCathodeVal:= 1E-5,
		ePumpStationPirani1State:= E_PressureState.ValidLo,
		ePumpStationPirani2State:= E_PressureState.ValidLo,
		fPumpStationColdCathodeVal:= 1E-5
	);
	stGaugeReadingsOp : ST_SBGaugeReadingsOp := (
		eDPPiraniOp:= E_GaugeCompOp.STATE, 
		eDPColdCathodeOp:= E_GaugeCompOp._LTE, 
		ePumpStationPirani1Op:= E_GaugeCompOp.STATE, 
		ePumpStationPirani2Op:= E_GaugeCompOp.STATE, 
		ePumpStationColdCathodeOp:= E_GaugeCompOp._LTE);
		
	stExpTTStatus : ST_TransportTubeStatuses := (bGateValveOpen:= FALSE);
	stTTOp : ST_TransportTubeOps := (bIonPumpIgnore:= TRUE);
		
	(* Expected system states after operation finishes *)
	stFinExpPumpStatus : ST_SBPumpStatuses := (
		bRoughingPumpOn:= FALSE, 
		bTurboPumpOn:= FALSE, 
		bIonPumpOn:= FALSE);
	
	stFinExpValveStatus : ST_SBValveStatuses := (
		bGateValveOpen:= FALSE, 
		bVentValveOpen:= FALSE, 
		bORingPumpValveOpen:= FALSE, 
		bForelineValveOpen:= FALSE, 
		bSlowPumpValveOpen:= FALSE,
		bSBVentOpen:= FALSE,  
		bSBSlowVentOpen:= FALSE);
	
	stFinExpGaugeReadings : ST_SBGaugeReadings := (
		eDPColdCathodeState := E_PressureState.Off,
		ePumpStationColdCathodeState := E_PressureState.Off
	);
	stFinGaugeReadingsOp : ST_SBGaugeReadingsOp := (
		eDPPiraniOp:= E_GaugeCompOp.ATM, 
		eDPColdCathodeOp:= E_GaugeCompOp.STATE, 
		ePumpStationPirani1Op:= E_GaugeCompOp.ATM, 
		ePumpStationPirani2Op:= E_GaugeCompOp.ATM, 
		ePumpStationColdCathodeOp:= E_GaugeCompOp.STATE);
		
	stFinExpTTStatus : ST_TransportTubeStatuses := (bGateValveOpen:= FALSE);
	stFinTTOp : ST_TransportTubeOps := (bIonPumpIgnore:= TRUE);
		
	(* Timeout constants *)
	VENT_TIMEOUT : TIME := T#10M;
	SLOW_VENT_TIMEOUT : TIME := T#30M;
	
	(* Pressure constants *)
	SLOW_VENT_PRESS : REAL := 1E-2; // Pressure (Torr) at which to begin slow venting
END_VAR

SUPER^(iq_sMessageBuffer := iq_sMessageBuffer);

CASE eStep OF
E_OpStep.IDLE: // Do nothing

E_OpStep.START: // Verify system status
	M_RunTimeoutTimer(STATUS_CHECK_TIMEOUT);
	M_SetMessage('Verifying system status');
	
	IF F_VerifySBPumpStatuses(stExpStatus := stExpPumpStatus, bEnforce := TRUE)
		AND F_VerifySBValveStatuses(stExpStatus := stExpValveStatus, bEnforce := TRUE)
		AND F_VerifySBGaugeReadings(stExpReadings := stExpGaugeReadings, stReadingsOp := stGaugeReadingsOp)
		AND F_VerifyAllTransportTubeStatuses(stExpStatus := stExpTTStatus, 
			stStatusOp := stTTOp,
			bEnforce := TRUE)
	THEN // System status check 
		M_ResetTimeoutTimer();
		M_SetMessage('Closing gate valve');
		eStep := E_OpStep.SVSB_CLOSE_GATE_VALVE;
	END_IF
	
E_OpStep.SVSB_CLOSE_GATE_VALVE:
	M_RunTimeoutTimer(VALVE_TIMEOUT);
	
	// Close gate valve to pump station to isolate pumps
	GVL_BTS_VAC.fb_PP_VGC.M_Set_OPN_SW(FALSE);
	
	IF GVL_BTS_VAC.fb_PP_VGC.M_IsClosed() THEN
		M_ResetTimeoutTimer();
		M_SetMessage('Closing foreline valve');
		eStep := E_OpStep.SVSB_CLOSE_FORELINE_VALVE;
	END_IF
	
E_OpStep.SVSB_CLOSE_FORELINE_VALVE:
	M_RunTimeoutTimer(VALVE_TIMEOUT);
	
	// Close valves to pumping station to isolate pumps
	GVL_BTS_VAC.fb_PP_VRC_2.M_Set_OPN_SW(FALSE);
	
	IF GVL_BTS_VAC.fb_PP_VRC_2.iq_stValve.eState = E_ValvePositionState.CLOSED THEN
		M_ResetTimeoutTimer();
		M_SetMessage('Turning off roughing and ion pump');
		eStep := E_OpStep.SVSB_TURN_OFF_PUMPS;
	END_IF
	
E_OpStep.SVSB_TURN_OFF_PUMPS:
	M_RunTimeoutTimer(PUMP_TIMEOUT);
	
	// Turn off pumping station pumps
	GVL_BTS_VAC.fb_PP_PMF.M_Run(FALSE);
	GVL_BTS_VAC.fb_PP_PIP.M_Run(FALSE);
	
	IF GVL_BTS_VAC.fb_PP_PMF.q_stPump.eState = E_PumpState.pumpSTOPPED AND NOT GVL_BTS_VAC.fb_PP_PIP.stPump.i_xSP_DI THEN
		M_ResetTimeoutTimer();
		M_SetMessage('Closing O-Ring valve');
		eStep := E_OpStep.SVSB_CLOSE_ORING_VALVE;
	END_IF
	
E_OpStep.SVSB_CLOSE_ORING_VALVE:
	M_RunTimeoutTimer(VALVE_TIMEOUT);
	
	// Close O-Ring pump valve
	GVL_BTS_VAC.fb_PP_VRC_1.M_Set_OPN_SW(FALSE);

	IF GVL_BTS_VAC.fb_PP_VRC_1.iq_stValve.eState = E_ValvePositionState.CLOSED THEN
		M_ResetTimeoutTimer();
		M_SetMessage('Venting');
		eStep := E_OpStep.SVSB_VENT;
	END_IF
	
E_OpStep.SVSB_VENT:
	M_RunTimeoutTimer(VENT_TIMEOUT);
		
	// Open switchbox vent
	GVL_BTS_VAC.fb_VP_VVC_1.M_Close(FALSE);
	
	// Vent until safe for slow vent
	IF GVL_BTS_VAC.fb_DP_GPI.PG.rPRESS >= SLOW_VENT_PRESS THEN
		M_ResetTimeoutTimer();
		M_SetMessage('Slow venting');
		eStep := E_OpStep.SVSB_SLOW_VENT;
	END_IF
	

E_OpStep.SVSB_SLOW_VENT:
	M_RunTimeoutTimer(SLOW_VENT_TIMEOUT);
	
	// Close main vent
	GVL_BTS_VAC.fb_VP_VVC_1.M_Close(TRUE);
	
	// Open slow vent
	GVL_BTS_VAC.fb_VP_VVC_2.M_Close(FALSE);
	
	// Vent till atmospheric pressure reached
	IF F_ATM(GVL_BTS_VAC.fb_DP_GPI.PG.rPRESS) THEN
		M_ResetTimeoutTimer();
		M_SetMessage('Closing vent');
		eStep := E_OpStep.SVSB_CLOSE_VENT;
	END_IF
	
E_OpStep.SVSB_CLOSE_VENT:
	GVL_BTS_VAC.fb_VP_VVC_2.M_Close(TRUE);
	// How to verfiy the vent is closed?
	eStep := E_OpStep.SVSB_FINISH;
	
E_OpStep.SVSB_FINISH:
	IF F_VerifySBPumpStatuses(stExpStatus := stFinExpPumpStatus, bEnforce := FALSE)
		AND F_VerifySBValveStatuses(stExpStatus := stFinExpValveStatus, bEnforce := FALSE)
		AND F_VerifySBGaugeReadings(stExpReadings := stFinExpGaugeReadings, stReadingsOp := stFinGaugeReadingsOp)
		AND F_VerifyAllTransportTubeStatuses(stExpStatus := stFinExpTTStatus, 
			stStatusOp := stFinTTOp,
			bEnforce := FALSE)
	THEN
		M_Finish();
	ELSE
		M_FatalError('End system status check failed');
	END_IF
	
ELSE
	M_FatalError('Operation is in invalid state');
END_CASE

END_FUNCTION_BLOCK

// ---- POUs/MaintainLaser.TcPOU
(* The job of FB_LaserMaintainer is to keep the LASER_OK signal for each
transport tube on for as long as safely possible. This involves shutting down
lasers for tubes that do not meet system status checks and switching out
failed pumps when necessary *)
PROGRAM MaintainLaser
VAR_TEMP
	bSwitchboxStatusOk : BOOL;
	nIter : UINT;
	eTT : T_TransportTube;
	fbTT : REFERENCE TO FB_TransportTube;
	nPumpFailures : UINT;
END_VAR
VAR
	fbSBIonPumpFailure : FB_SwitchboxIonPumpFailure;
	fbSBRoughingOrTurboPumpFailure : FB_SwitchboxRoughingOrTurboPumpFailure;
END_VAR
VAR CONSTANT
	stExpValveStatus : ST_SBValveStatuses := (
		bGateValveOpen:= FALSE, 
		bVentValveOpen:= FALSE, 
		bORingPumpValveOpen:= TRUE, 
		bForelineValveOpen:= TRUE, 
		bSlowPumpValveOpen:= FALSE,
		bSBVentOpen:= FALSE,  
		bSBSlowVentOpen:= FALSE);
	
	stExpGaugeReadings : ST_SBGaugeReadings := (
		eDPPiraniState:= E_PressureState.ValidLo,
		fDPColdCathodeVal:= 1E-5,
		ePumpStationPirani1State:= E_PressureState.ValidLo,
		fPumpStationPirani2Val:= 1E-2,
		fPumpStationColdCathodeVal:= 1E-5
	);
	stGaugeReadingsOp : ST_SBGaugeReadingsOp := (
		eDPPiraniOp:= E_GaugeCompOp.STATE, 
		eDPColdCathodeOp:= E_GaugeCompOp._LTE, 
		ePumpStationPirani1Op:= E_GaugeCompOp.STATE, 
		ePumpStationPirani2Op:= E_GaugeCompOp._LTE, 
		ePumpStationColdCathodeOp:= E_GaugeCompOp._LTE);
		
	stExpTTStatus : ST_TransportTubeStatuses := (
		bIonPumpOn:= TRUE,
		bGateValveOpen:= TRUE,
		ePiraniState:= E_PressureState.ValidLo,
		fColdCathodeVal:= 1E-5);
	stTTOp : ST_TransportTubeOps := (
		ePiraniOp := E_GaugeCompOp.STATE,
		eColdCathodeOp := E_GaugeCompOp._LTE
	);
END_VAR

IF GVL_MaintainLaser.i_bReset THEN
	GVL_MaintainLaser.q_bIonPumpFailure := FALSE;
	GVL_MaintainLaser.q_bRoughingPumpFailure := FALSE;
	GVL_MaintainLaser.q_bTurboPumpFailure := FALSE;
	
	fbSBIonPumpFailure(i_bExecute := FALSE, 
						i_bCancel := TRUE, 
						iq_sMessageBuffer := GVL_MaintainLaser.q_sMessage);
	fbSBIonPumpFailure.M_ResetError();
	
	fbSBRoughingOrTurboPumpFailure(i_bExecute := FALSE,
									i_bCancel := TRUE, 
									iq_sMessageBuffer := GVL_MaintainLaser.q_sMessage);
	fbSBRoughingOrTurboPumpFailure.M_ResetError();
	GVL_MaintainLaser.q_sMessage := 'No issues';
	
	GVL_MaintainLaser.q_bOperationInProgress := FALSE;
	GVL_MaintainLaser.i_bShutoff := FALSE;
	GVL_MaintainLaser.i_bReset := FALSE;
	GVL_MaintainLaser.q_bShutoffLatch := FALSE;
END_IF

// Look for pump failures. Once a pump failure is detected, latch the error until reset
GVL_MaintainLaser.q_bIonPumpFailure := GVL_MaintainLaser.q_bIonPumpFailure OR TRUE; // TODO, figure out how  check for ion pump failure
GVL_MaintainLaser.q_bTurboPumpFailure := GVL_MaintainLaser.q_bTurboPumpFailure OR GVL_BTS_VAC.fb_PP_PTM.iq_stPTM.eState = E_PumpState.pumpFAULT;
GVL_MaintainLaser.q_bRoughingPumpFailure := GVL_MaintainLaser.q_bRoughingPumpFailure OR GVL_BTS_VAC.fb_PP_PMF.q_stPump.eState = E_PumpState.pumpFAULT;

// Count the number of pump failures
nPumpFailures := BOOL_TO_UINT(GVL_MaintainLaser.q_bTurboPumpFailure) + BOOL_TO_UINT(GVL_MaintainLaser.q_bIonPumpFailure) + BOOL_TO_UINT(GVL_MaintainLaser.q_bRoughingPumpFailure);

// If a pump failure accured. Attempt to maintain vacuum as long as possible. If there are multiple pump failures then the system is not recoverable.
// Once a recovery operation has finished with an error or a shutdown laser signal, keep it from re-running until reset.
fbSBIonPumpFailure(i_bExecute := nPumpFailures = 1 
		AND GVL_MaintainLaser.q_bIonPumpFailure 
		AND NOT fbSBIonPumpFailure.q_bError 
		AND NOT fbSBIonPumpFailure.q_bShutdownLaser,
	i_bCancel := FALSE,
	iq_sMessageBuffer := GVL_MaintainLaser.q_sMessage);
fbSBRoughingOrTurboPumpFailure(i_bExecute := nPumpFailures = 1 
		AND (GVL_MaintainLaser.q_bRoughingPumpFailure OR GVL_MaintainLaser.q_bTurboPumpFailure) 
		AND NOT fbSBRoughingOrTurboPumpFailure.q_bError 
		AND NOT fbSBRoughingOrTurboPumpFailure.q_bShutdownLaser,
	i_bCancel := FALSE,
	iq_sMessageBuffer := GVL_MaintainLaser.q_sMessage);

GVL_MaintainLaser.q_bOperationInProgress := fbSBIonPumpFailure.q_bBusy OR fbSBRoughingOrTurboPumpFailure.q_bBusy;

(* Verify the switchbox is in an okay state for lasers. *)
bSwitchboxStatusOk :=
	nPumpFailures <= 1
	AND NOT fbSBIonPumpFailure.q_bShutdownLaser
	AND NOT fbSBRoughingOrTurboPumpFailure.q_bShutdownLaser;

(* Additional checks for switchbox for when there is not a pump failure. When a pump failure happens, these checks are no longer valid *)
IF nPumpFailures = 0 THEN
	bSwitchboxStatusOk := F_VerifySBValveStatuses(stExpStatus := stExpValveStatus, bEnforce := FALSE)
		AND F_VerifySBGaugeReadings(stExpReadings := stExpGaugeReadings, stReadingsOp := stGaugeReadingsOp);
END_IF

